LIN {X 0,Y 115.253,Z 407.117,A -85,B 0,C 180,E1 -25932.672,E2 -25932.672} C_VEL
LIN {X 0,Y 115.008,Z 407.148,A -85,B 0,C 180,E1 -25937.79,E2 -25937.79} C_VEL
LIN {X 0,Y 114.944,Z 407.16,A -85,B 0,C 180,E1 -25943.492,E2 -25943.492} C_VEL
LIN {X 0,Y 114.866,Z 407.178,A -85,B 0,C 180,E1 -25946.088,E2 -25946.088} C_VEL
LIN {X 0,Y 115.76,Z 409.771,A -85,B 0,C 180,E1 -25947.086,E2 -25947.086} C_VEL
LIN {X 0,Y 117.751,Z 412.046,A -85,B 0,C 180,E1 -25948.695,E2 -25948.695} C_VEL
LIN {X 0,Y 118.702,Z 412.889,A -85,B 0,C 180,E1 -25949.4,E2 -25949.4} C_VEL
LIN {X 0,Y 120.73,Z 416.135,A -85,B 0,C 180,E1 -25950.969,E2 -25950.969} C_VEL
LIN {X 0,Y 122.361,Z 417.964,A -85,B 0,C 180,E1 -25952.092,E2 -25952.092} C_VEL
LIN {X 0,Y 128.066,Z 426.389,A -85,B 0,C 180,E1 -25955.788,E2 -25955.788} C_VEL
LIN {X 0,Y 130.824,Z 431.068,A -85,B 0,C 180,E1 -25957.424,E2 -25957.424} C_VEL
LIN {X 0,Y 135.904,Z 442.797,A -85,B 0,C 180,E1 -25960.392,E2 -25960.392} C_VEL
LIN {X 0,Y 139.945,Z 454.557,A -85,B 0,C 180,E1 -25962.684,E2 -25962.684} C_VEL
LIN {X 0,Y 140.862,Z 457.48,A -85,B 0,C 180,E1 -25963.193,E2 -25963.193} C_VEL
LIN {X 0,Y 141.678,Z 474.746,A -85,B 0,C 180,E1 -25964.592,E2 -25964.592} C_VEL
LIN {X 0,Y 139.119,Z 511.457,A -85,B 0,C 180,E1 -25966.251,E2 -25966.251} C_VEL
LIN {X 0,Y 137.344,Z 525.013,A -85,B 0,C 180,E1 -25967.355,E2 -25967.355} C_VEL
LIN {X 0,Y 134.916,Z 537.503,A -85,B 0,C 180,E1 -25968.88,E2 -25968.88} C_VEL
LIN {X 0,Y 132.501,Z 547.084,A -85,B 0,C 180,E1 -25970.47,E2 -25970.47} C_VEL
LIN {X 0,Y 129.221,Z 557.848,A -85,B 0,C 180,E1 -25972.768,E2 -25972.768} C_VEL
LIN {X 0,Y 126.712,Z 565.45,A -85,B 0,C 180,E1 -25974.87,E2 -25974.87} C_VEL
LIN {X 0,Y 123.341,Z 575.06,A -85,B 0,C 180,E1 -25978.193,E2 -25978.193} C_VEL
LIN {X 0,Y 119.874,Z 583.772,A -85,B 0,C 180,E1 -25982.03,E2 -25982.03} C_VEL
LIN {X 0,Y 117.346,Z 591.006,A -85,B 0,C 180,E1 -25986.156,E2 -25986.156} C_VEL
LIN {X 0,Y 114.881,Z 598.038,A -85,B 0,C 180,E1 -25991.266,E2 -25991.266} C_VEL
LIN {X 0,Y 113.15,Z 604.474,A -85,B 0,C 180,E1 -25997.444,E2 -25997.444} C_VEL
LIN {X 0,Y 112.538,Z 608.664,A -85,B 0,C 180,E1 -26002.825,E2 -26002.825} C_VEL
LIN {X 0,Y 112.496,Z 611.794,A -85,B 0,C 180,E1 -26008.312,E2 -26008.312} C_VEL
LIN {X 0,Y 112.529,Z 613.372,A -85,B 0,C 180,E1 -26012.193,E2 -26012.193} C_VEL
LIN {X 0,Y 112.474,Z 614.612,A -85,B 0,C 180,E1 -26017.179,E2 -26017.179} C_VEL
LIN {X 0,Y 112.828,Z 615.053,A -85,B 0,C 180,E1 -26020.77,E2 -26020.77} C_VEL
LIN {X 0,Y 114.707,Z 614.724,A -85,B 0,C 180,E1 -26027.839,E2 -26027.839} C_VEL
LIN {X 0,Y 118.407,Z 612.906,A -85,B 0,C 180,E1 -26034.549,E2 -26034.549} C_VEL
LIN {X 0,Y 120.829,Z 611.384,A -85,B 0,C 180,E1 -26037.73,E2 -26037.73} C_VEL
LIN {X 0,Y 125.198,Z 608.337,A -85,B 0,C 180,E1 -26042.227,E2 -26042.227} C_VEL
LIN {X 0,Y 130.219,Z 604.271,A -85,B 0,C 180,E1 -26046.417,E2 -26046.417} C_VEL
LIN {X 0,Y 136.995,Z 598.08,A -85,B 0,C 180,E1 -26050.849,E2 -26050.849} C_VEL
LIN {X 0,Y 143.504,Z 591.376,A -85,B 0,C 180,E1 -26054.256,E2 -26054.256} C_VEL
LIN {X 0,Y 150.582,Z 583.094,A -85,B 0,C 180,E1 -26057.313,E2 -26057.313} C_VEL
LIN {X 0,Y 157.336,Z 573.799,A -85,B 0,C 180,E1 -26059.829,E2 -26059.829} C_VEL
LIN {X 0,Y 159.711,Z 569.48,A -85,B 0,C 180,E1 -26060.999,E2 -26060.999} C_VEL
LIN {X 0,Y 162.549,Z 562.182,A -85,B 0,C 180,E1 -26063.181,E2 -26063.181} C_VEL
LIN {X 0,Y 165.228,Z 554.511,A -85,B 0,C 180,E1 -26065.144,E2 -26065.144} C_VEL
LIN {X 0,Y 167.258,Z 549.517,A -85,B 0,C 180,E1 -26065.962,E2 -26065.962} C_VEL
LIN {X 0,Y 171.699,Z 538.632,A -85,B 0,C 180,E1 -26067.044,E2 -26067.044} C_VEL
LIN {X 0,Y 175.674,Z 525.948,A -85,B 0,C 180,E1 -26067.969,E2 -26067.969} C_VEL
LIN {X 0,Y 178.474,Z 513.103,A -85,B 0,C 180,E1 -26068.575,E2 -26068.575} C_VEL
LIN {X 0,Y 180.148,Z 498.961,A -85,B 0,C 180,E1 -26069.084,E2 -26069.084} C_VEL
LIN {X 0,Y 177.319,Z 490.638,A -85,B 0,C 180,E1 -26072.157,E2 -26072.157} C_VEL
LIN {X 0,Y 175.145,Z 484.92,A -85,B 0,C 180,E1 -26074.844,E2 -26074.844} C_VEL
LIN {X 0,Y 173.289,Z 480.416,A -85,B 0,C 180,E1 -26077.496,E2 -26077.496} C_VEL
LIN {X 0,Y 172.175,Z 477.636,A -85,B 0,C 180,E1 -26079.409,E2 -26079.409} C_VEL
LIN {X 0,Y 170.647,Z 473.807,A -85,B 0,C 180,E1 -26082.724,E2 -26082.724} C_VEL
LIN {X 0,Y 168.918,Z 469.43,A -85,B 0,C 180,E1 -26089.548,E2 -26089.548} C_VEL
LIN {X 0,Y 169.073,Z 469.433,A -85,B 0,C 180,E1 -26096.032,E2 -26096.032} C_VEL
LIN {X 0,Y 170.368,Z 472.982,A -85,B 0,C 180,E1 -26101.182,E2 -26101.182} C_VEL
LIN {X 0,Y 171.205,Z 474.143,A -85,B 0,C 180,E1 -26103.053,E2 -26103.053} C_VEL
LIN {X 0,Y 173.451,Z 478.47,A -85,B 0,C 180,E1 -26107.09,E2 -26107.09} C_VEL
LIN {X 0,Y 175.519,Z 482.29,A -85,B 0,C 180,E1 -26109.871,E2 -26109.871} C_VEL
LIN {X 0,Y 177.675,Z 486.397,A -85,B 0,C 180,E1 -26112.348,E2 -26112.348} C_VEL
LIN {X 0,Y 180.685,Z 492.68,A -85,B 0,C 180,E1 -26115.367,E2 -26115.367} C_VEL
LIN {X 0,Y 178.925,Z 507.485,A -85,B 0,C 180,E1 -26115.96,E2 -26115.96} C_VEL
LIN {X 0,Y 176.106,Z 520.316,A -85,B 0,C 180,E1 -26116.712,E2 -26116.712} C_VEL
LIN {X 0,Y 172.039,Z 533.167,A -85,B 0,C 180,E1 -26117.764,E2 -26117.764} C_VEL
LIN {X 0,Y 167.387,Z 544.658,A -85,B 0,C 180,E1 -26119.152,E2 -26119.152} C_VEL
LIN {X 0,Y 161.724,Z 555.648,A -85,B 0,C 180,E1 -26120.885,E2 -26120.885} C_VEL
LIN {X 0,Y 155.509,Z 565.605,A -85,B 0,C 180,E1 -26122.957,E2 -26122.957} C_VEL
LIN {X 0,Y 149.551,Z 573.711,A -85,B 0,C 180,E1 -26125.184,E2 -26125.184} C_VEL
LIN {X 0,Y 143.124,Z 581.245,A -85,B 0,C 180,E1 -26127.889,E2 -26127.889} C_VEL
LIN {X 0,Y 137.04,Z 587.443,A -85,B 0,C 180,E1 -26130.855,E2 -26130.855} C_VEL
LIN {X 0,Y 131.424,Z 592.438,A -85,B 0,C 180,E1 -26134.019,E2 -26134.019} C_VEL
LIN {X 0,Y 125.209,Z 597.266,A -85,B 0,C 180,E1 -26138.205,E2 -26138.205} C_VEL
LIN {X 0,Y 119.698,Z 600.886,A -85,B 0,C 180,E1 -26142.784,E2 -26142.784} C_VEL
LIN {X 0,Y 114.942,Z 603.398,A -85,B 0,C 180,E1 -26147.734,E2 -26147.734} C_VEL
LIN {X 0,Y 112.305,Z 604.491,A -85,B 0,C 180,E1 -26151.261,E2 -26151.261} C_VEL
LIN {X 0,Y 109.04,Z 605.323,A -85,B 0,C 180,E1 -26156.921,E2 -26156.921} C_VEL
LIN {X 0,Y 106.781,Z 605.183,A -85,B 0,C 180,E1 -26162.567,E2 -26162.567} C_VEL
LIN {X 0,Y 105.395,Z 603.928,A -85,B 0,C 180,E1 -26169,E2 -26169} C_VEL
LIN {X 0,Y 104.928,Z 602.013,A -85,B 0,C 180,E1 -26174.46,E2 -26174.46} C_VEL
LIN {X 0,Y 105.341,Z 598.939,A -85,B 0,C 180,E1 -26180.399,E2 -26180.399} C_VEL
LIN {X 0,Y 106.568,Z 594.793,A -85,B 0,C 180,E1 -26186.219,E2 -26186.219} C_VEL
LIN {X 0,Y 108.751,Z 588.456,A -85,B 0,C 180,E1 -26192.778,E2 -26192.778} C_VEL
LIN {X 0,Y 111.475,Z 581.569,A -85,B 0,C 180,E1 -26198.155,E2 -26198.155} C_VEL
LIN {X 0,Y 114.368,Z 574.542,A -85,B 0,C 180,E1 -26202.42,E2 -26202.42} C_VEL
LIN {X 0,Y 117.794,Z 565.906,A -85,B 0,C 180,E1 -26206.552,E2 -26206.552} C_VEL
LIN {X 0,Y 121.146,Z 556.837,A -85,B 0,C 180,E1 -26209.927,E2 -26209.927} C_VEL
LIN {X 0,Y 125.019,Z 545.291,A -85,B 0,C 180,E1 -26213.172,E2 -26213.172} C_VEL
LIN {X 0,Y 128.216,Z 533.972,A -85,B 0,C 180,E1 -26215.572,E2 -26215.572} C_VEL
LIN {X 0,Y 130.805,Z 522.488,A -85,B 0,C 180,E1 -26217.39,E2 -26217.39} C_VEL
LIN {X 0,Y 133.005,Z 509.199,A -85,B 0,C 180,E1 -26218.844,E2 -26218.844} C_VEL
LIN {X 0,Y 134.384,Z 495.992,A -85,B 0,C 180,E1 -26219.741,E2 -26219.741} C_VEL
LIN {X 0,Y 137.172,Z 456.576,A -85,B 0,C 180,E1 -26221.49,E2 -26221.49} C_VEL
LIN {X 0,Y 131.241,Z 443.73,A -85,B 0,C 180,E1 -26224.758,E2 -26224.758} C_VEL
LIN {X 0,Y 125.369,Z 433.254,A -85,B 0,C 180,E1 -26228.294,E2 -26228.294} C_VEL
LIN {X 0,Y 120.436,Z 425.822,A -85,B 0,C 180,E1 -26231.61,E2 -26231.61} C_VEL
LIN {X 0,Y 118.211,Z 422.576,A -85,B 0,C 180,E1 -26233.267,E2 -26233.267} C_VEL
LIN {X 0,Y 115.739,Z 419.077,A -85,B 0,C 180,E1 -26235.249,E2 -26235.249} C_VEL
LIN {X 0,Y 112.788,Z 415.592,A -85,B 0,C 180,E1 -26237.794,E2 -26237.794} C_VEL
LIN {X 0,Y 111.683,Z 413.593,A -85,B 0,C 180,E1 -26238.914,E2 -26238.914} C_VEL
LIN {X 0,Y 109.275,Z 411.704,A -85,B 0,C 180,E1 -26241.243,E2 -26241.243} C_VEL
LIN {X 0,Y 108.072,Z 409.461,A -85,B 0,C 180,E1 -26242.688,E2 -26242.688} C_VEL
LIN {X 0,Y 107.728,Z 408.052,A -85,B 0,C 180,E1 -26243.368,E2 -26243.368} C_VEL
LIN {X 0,Y 107.799,Z 408.044,A -85,B 0,C 180,E1 -26248.562,E2 -26248.562} C_VEL
LIN {X 0,Y 107.91,Z 408.028,A -85,B 0,C 180,E1 -26256.996,E2 -26256.996} C_VEL
LIN {X 0,Y 108.027,Z 408.014,A -85,B 0,C 180,E1 -26264.915,E2 -26264.915} C_VEL
LIN {X 0,Y 108.254,Z 407.99,A -85,B 0,C 180,E1 -26268.768,E2 -26268.768} C_VEL
LIN {X 0,Y 108.444,Z 407.964,A -85,B 0,C 180,E1 -26276.283,E2 -26276.283} C_VEL
LIN {X 0,Y 108.915,Z 407.86,A -85,B 0,C 180,E1 -26279.999,E2 -26279.999} C_VEL
LIN {X 0,Y 108.301,Z 407.991,A -85,B 0,C 180,E1 -26287.456,E2 -26287.456} C_VEL
LIN {X 0,Y 108.173,Z 408,A -85,B 0,C 180,E1 -26292.959,E2 -26292.959} C_VEL
LIN {X 0,Y 107.943,Z 408.218,A -85,B 0,C 180,E1 -26300.359,E2 -26300.359} C_VEL
LIN {X 0,Y 108.73,Z 410.548,A -85,B 0,C 180,E1 -26301.444,E2 -26301.444} C_VEL
LIN {X 0,Y 110.675,Z 412.834,A -85,B 0,C 180,E1 -26303.485,E2 -26303.485} C_VEL
LIN {X 0,Y 112.053,Z 413.96,A -85,B 0,C 180,E1 -26304.763,E2 -26304.763} C_VEL
LIN {X 0,Y 114.154,Z 417.301,A -85,B 0,C 180,E1 -26306.756,E2 -26306.756} C_VEL
LIN {X 0,Y 115.855,Z 419.178,A -85,B 0,C 180,E1 -26308.165,E2 -26308.165} C_VEL
LIN {X 0,Y 118.456,Z 422.775,A -85,B 0,C 180,E1 -26310.232,E2 -26310.232} C_VEL
LIN {X 0,Y 122.616,Z 428.986,A -85,B 0,C 180,E1 -26313.236,E2 -26313.236} C_VEL
LIN {X 0,Y 126.523,Z 435.357,A -85,B 0,C 180,E1 -26315.786,E2 -26315.786} C_VEL
LIN {X 0,Y 131.342,Z 446.96,A -85,B 0,C 180,E1 -26318.864,E2 -26318.864} C_VEL
LIN {X 0,Y 135.02,Z 458.215,A -85,B 0,C 180,E1 -26321.159,E2 -26321.159} C_VEL
LIN {X 0,Y 135.529,Z 460.494,A -85,B 0,C 180,E1 -26321.512,E2 -26321.512} C_VEL
LIN {X 0,Y 136.182,Z 474.785,A -85,B 0,C 180,E1 -26322.748,E2 -26322.748} C_VEL
LIN {X 0,Y 133.574,Z 510.886,A -85,B 0,C 180,E1 -26324.416,E2 -26324.416} C_VEL
LIN {X 0,Y 131.674,Z 524.54,A -85,B 0,C 180,E1 -26325.531,E2 -26325.531} C_VEL
LIN {X 0,Y 129.103,Z 537.266,A -85,B 0,C 180,E1 -26327.121,E2 -26327.121} C_VEL
LIN {X 0,Y 126.576,Z 546.828,A -85,B 0,C 180,E1 -26328.751,E2 -26328.751} C_VEL
LIN {X 0,Y 123.147,Z 557.577,A -85,B 0,C 180,E1 -26331.115,E2 -26331.115} C_VEL
LIN {X 0,Y 120.493,Z 565.166,A -85,B 0,C 180,E1 -26333.285,E2 -26333.285} C_VEL
LIN {X 0,Y 117.302,Z 573.776,A -85,B 0,C 180,E1 -26336.345,E2 -26336.345} C_VEL
LIN {X 0,Y 114.329,Z 580.973,A -85,B 0,C 180,E1 -26339.503,E2 -26339.503} C_VEL
LIN {X 0,Y 111.365,Z 588.648,A -85,B 0,C 180,E1 -26343.785,E2 -26343.785} C_VEL
LIN {X 0,Y 108.54,Z 596.111,A -85,B 0,C 180,E1 -26349.138,E2 -26349.138} C_VEL
LIN {X 0,Y 106.591,Z 602.073,A -85,B 0,C 180,E1 -26354.708,E2 -26354.708} C_VEL
LIN {X 0,Y 105.642,Z 606.757,A -85,B 0,C 180,E1 -26360.426,E2 -26360.426} C_VEL
LIN {X 0,Y 105.39,Z 610.28,A -85,B 0,C 180,E1 -26366.176,E2 -26366.176} C_VEL
LIN {X 0,Y 105.548,Z 612.037,A -85,B 0,C 180,E1 -26370,E2 -26370} C_VEL
LIN {X 0,Y 105.389,Z 613.311,A -85,B 0,C 180,E1 -26373.824,E2 -26373.824} C_VEL
LIN {X 0,Y 105.834,Z 614.67,A -85,B 0,C 180,E1 -26381.491,E2 -26381.491} C_VEL
LIN {X 0,Y 106.688,Z 614.76,A -85,B 0,C 180,E1 -26385.277,E2 -26385.277} C_VEL
LIN {X 0,Y 109.705,Z 613.761,A -85,B 0,C 180,E1 -26392.605,E2 -26392.605} C_VEL
LIN {X 0,Y 114.575,Z 611.256,A -85,B 0,C 180,E1 -26399.387,E2 -26399.387} C_VEL
LIN {X 0,Y 119.817,Z 607.841,A -85,B 0,C 180,E1 -26404.603,E2 -26404.603} C_VEL
LIN {X 0,Y 126.503,Z 602.701,A -85,B 0,C 180,E1 -26409.708,E2 -26409.708} C_VEL
LIN {X 0,Y 133.931,Z 596.208,A -85,B 0,C 180,E1 -26414.049,E2 -26414.049} C_VEL
LIN {X 0,Y 140.938,Z 589.139,A -85,B 0,C 180,E1 -26417.35,E2 -26417.35} C_VEL
LIN {X 0,Y 148.421,Z 580.361,A -85,B 0,C 180,E1 -26420.305,E2 -26420.305} C_VEL
LIN {X 0,Y 155.615,Z 570.432,A -85,B 0,C 180,E1 -26422.747,E2 -26422.747} C_VEL
LIN {X 0,Y 161.818,Z 560.324,A -85,B 0,C 180,E1 -26424.52,E2 -26424.52} C_VEL
LIN {X 0,Y 167.258,Z 549.517,A -85,B 0,C 180,E1 -26425.962,E2 -26425.962} C_VEL
LIN {X 0,Y 169.166,Z 544.407,A -85,B 0,C 180,E1 -26426.717,E2 -26426.717} C_VEL
LIN {X 0,Y 171.161,Z 535.908,A -85,B 0,C 180,E1 -26428.307,E2 -26428.307} C_VEL
LIN {X 0,Y 172.711,Z 527.169,A -85,B 0,C 180,E1 -26429.764,E2 -26429.764} C_VEL
LIN {X 0,Y 173.83,Z 521.619,A -85,B 0,C 180,E1 -26430.314,E2 -26430.314} C_VEL
LIN {X 0,Y 176.309,Z 508.882,A -85,B 0,C 180,E1 -26430.844,E2 -26430.844} C_VEL
LIN {X 0,Y 177.063,Z 502.166,A -85,B 0,C 180,E1 -26431.088,E2 -26431.088} C_VEL
LIN {X 0,Y 174.716,Z 494.887,A -85,B 0,C 180,E1 -26433.979,E2 -26433.979} C_VEL
LIN {X 0,Y 172.504,Z 488.69,A -85,B 0,C 180,E1 -26437.151,E2 -26437.151} C_VEL
LIN {X 0,Y 170.816,Z 484.212,A -85,B 0,C 180,E1 -26440.165,E2 -26440.165} C_VEL
LIN {X 0,Y 169.455,Z 480.555,A -85,B 0,C 180,E1 -26443.393,E2 -26443.393} C_VEL
LIN {X 0,Y 167.982,Z 476.435,A -85,B 0,C 180,E1 -26449.928,E2 -26449.928} C_VEL
LIN {X 0,Y 168.17,Z 476.581,A -85,B 0,C 180,E1 -26456.011,E2 -26456.011} C_VEL
LIN {X 0,Y 169.126,Z 479.622,A -85,B 0,C 180,E1 -26460.298,E2 -26460.298} C_VEL
LIN {X 0,Y 169.969,Z 480.84,A -85,B 0,C 180,E1 -26462.37,E2 -26462.37} C_VEL
LIN {X 0,Y 172,Z 485.034,A -85,B 0,C 180,E1 -26466.333,E2 -26466.333} C_VEL
LIN {X 0,Y 174.107,Z 489.188,A -85,B 0,C 180,E1 -26469.366,E2 -26469.366} C_VEL
LIN {X 0,Y 177.049,Z 495.311,A -85,B 0,C 180,E1 -26472.83,E2 -26472.83} C_VEL
LIN {X 0,Y 177.618,Z 496.635,A -85,B 0,C 180,E1 -26473.443,E2 -26473.443} C_VEL
LIN {X 0,Y 175.731,Z 509.626,A -85,B 0,C 180,E1 -26473.951,E2 -26473.951} C_VEL
LIN {X 0,Y 172.695,Z 522.371,A -85,B 0,C 180,E1 -26474.708,E2 -26474.708} C_VEL
LIN {X 0,Y 168.729,Z 534.274,A -85,B 0,C 180,E1 -26475.693,E2 -26475.693} C_VEL
LIN {X 0,Y 163.622,Z 546.148,A -85,B 0,C 180,E1 -26477.124,E2 -26477.124} C_VEL
LIN {X 0,Y 157.583,Z 557.253,A -85,B 0,C 180,E1 -26478.872,E2 -26478.872} C_VEL
LIN {X 0,Y 152.044,Z 565.713,A -85,B 0,C 180,E1 -26480.61,E2 -26480.61} C_VEL
LIN {X 0,Y 145.129,Z 574.749,A -85,B 0,C 180,E1 -26483.064,E2 -26483.064} C_VEL
LIN {X 0,Y 138.482,Z 582.111,A -85,B 0,C 180,E1 -26485.737,E2 -26485.737} C_VEL
LIN {X 0,Y 131.112,Z 589.093,A -85,B 0,C 180,E1 -26489.224,E2 -26489.224} C_VEL
LIN {X 0,Y 125.088,Z 594.012,A -85,B 0,C 180,E1 -26492.569,E2 -26492.569} C_VEL
LIN {X 0,Y 118.379,Z 598.69,A -85,B 0,C 180,E1 -26497.085,E2 -26497.085} C_VEL
LIN {X 0,Y 112.898,Z 601.877,A -85,B 0,C 180,E1 -26501.669,E2 -26501.669} C_VEL
LIN {X 0,Y 109.512,Z 603.507,A -85,B 0,C 180,E1 -26505.096,E2 -26505.096} C_VEL
LIN {X 0,Y 106.542,Z 604.699,A -85,B 0,C 180,E1 -26508.728,E2 -26508.728} C_VEL
LIN {X 0,Y 102.488,Z 605.665,A -85,B 0,C 180,E1 -26515.377,E2 -26515.377} C_VEL
LIN {X 0,Y 100.219,Z 605.582,A -85,B 0,C 180,E1 -26520.602,E2 -26520.602} C_VEL
LIN {X 0,Y 98.388,Z 604.245,A -85,B 0,C 180,E1 -26528.223,E2 -26528.223} C_VEL
LIN {X 0,Y 97.865,Z 602.604,A -85,B 0,C 180,E1 -26533.307,E2 -26533.307} C_VEL
LIN {X 0,Y 98.162,Z 599.637,A -85,B 0,C 180,E1 -26539.689,E2 -26539.689} C_VEL
LIN {X 0,Y 99.323,Z 595.612,A -85,B 0,C 180,E1 -26545.943,E2 -26545.943} C_VEL
LIN {X 0,Y 101.176,Z 590.451,A -85,B 0,C 180,E1 -26551.99,E2 -26551.99} C_VEL
LIN {X 0,Y 103.832,Z 583.961,A -85,B 0,C 180,E1 -26557.78,E2 -26557.78} C_VEL
LIN {X 0,Y 107.381,Z 575.844,A -85,B 0,C 180,E1 -26563.242,E2 -26563.242} C_VEL
LIN {X 0,Y 111.167,Z 566.932,A -85,B 0,C 180,E1 -26567.816,E2 -26567.816} C_VEL
LIN {X 0,Y 114.882,Z 557.497,A -85,B 0,C 180,E1 -26571.534,E2 -26571.534} C_VEL
LIN {X 0,Y 118.972,Z 546.031,A -85,B 0,C 180,E1 -26574.89,E2 -26574.89} C_VEL
LIN {X 0,Y 122.312,Z 534.816,A -85,B 0,C 180,E1 -26577.366,E2 -26577.366} C_VEL
LIN {X 0,Y 125.293,Z 522.284,A -85,B 0,C 180,E1 -26579.393,E2 -26579.393} C_VEL
LIN {X 0,Y 127.558,Z 509.173,A -85,B 0,C 180,E1 -26580.834,E2 -26580.834} C_VEL
LIN {X 0,Y 128.99,Z 495.882,A -85,B 0,C 180,E1 -26581.743,E2 -26581.743} C_VEL
LIN {X 0,Y 131.739,Z 458.836,A -85,B 0,C 180,E1 -26583.411,E2 -26583.411} C_VEL
LIN {X 0,Y 126.381,Z 447.016,A -85,B 0,C 180,E1 -26586.66,E2 -26586.66} C_VEL
LIN {X 0,Y 120.783,Z 436.959,A -85,B 0,C 180,E1 -26590.377,E2 -26590.377} C_VEL
LIN {X 0,Y 115.331,Z 428.518,A -85,B 0,C 180,E1 -26594.525,E2 -26594.525} C_VEL
LIN {X 0,Y 112.025,Z 424.051,A -85,B 0,C 180,E1 -26597.399,E2 -26597.399} C_VEL
LIN {X 0,Y 109.54,Z 420.544,A -85,B 0,C 180,E1 -26599.857,E2 -26599.857} C_VEL
LIN {X 0,Y 108.684,Z 419.589,A -85,B 0,C 180,E1 -26600.739,E2 -26600.739} C_VEL
LIN {X 0,Y 106.413,Z 417.142,A -85,B 0,C 180,E1 -26603.254,E2 -26603.254} C_VEL
LIN {X 0,Y 105.258,Z 414.722,A -85,B 0,C 180,E1 -26604.837,E2 -26604.837} C_VEL
LIN {X 0,Y 102.666,Z 412.959,A -85,B 0,C 180,E1 -26608.238,E2 -26608.238} C_VEL
LIN {X 0,Y 101.105,Z 410.644,A -85,B 0,C 180,E1 -26610.883,E2 -26610.883} C_VEL
LIN {X 0,Y 100.692,Z 408.94,A -85,B 0,C 180,E1 -26612.034,E2 -26612.034} C_VEL
LIN {X 0,Y 100.786,Z 408.917,A -85,B 0,C 180,E1 -26615.266,E2 -26615.266} C_VEL
LIN {X 0,Y 100.814,Z 408.926,A -85,B 0,C 180,E1 -26619.599,E2 -26619.599} C_VEL
LIN {X 0,Y 101.102,Z 408.888,A -85,B 0,C 180,E1 -26626.697,E2 -26626.697} C_VEL
LIN {X 0,Y 101.242,Z 408.858,A -85,B 0,C 180,E1 -26632.018,E2 -26632.018} C_VEL
LIN {X 0,Y 101.842,Z 408.739,A -85,B 0,C 180,E1 -26639.999,E2 -26639.999} C_VEL
LIN {X 0,Y 101.24,Z 408.873,A -85,B 0,C 180,E1 -26647.98,E2 -26647.98} C_VEL
LIN {X 0,Y 101.165,Z 408.908,A -85,B 0,C 180,E1 -26652.183,E2 -26652.183} C_VEL
LIN {X 0,Y 101.902,Z 411.444,A -85,B 0,C 180,E1 -26653.772,E2 -26653.772} C_VEL
LIN {X 0,Y 103.665,Z 413.707,A -85,B 0,C 180,E1 -26656.492,E2 -26656.492} C_VEL
LIN {X 0,Y 105.525,Z 414.848,A -85,B 0,C 180,E1 -26658.819,E2 -26658.819} C_VEL
LIN {X 0,Y 107.306,Z 418.07,A -85,B 0,C 180,E1 -26661.113,E2 -26661.113} C_VEL
LIN {X 0,Y 109.51,Z 420.308,A -85,B 0,C 180,E1 -26663.425,E2 -26663.425} C_VEL
LIN {X 0,Y 111.933,Z 423.843,A -85,B 0,C 180,E1 -26665.832,E2 -26665.832} C_VEL
LIN {X 0,Y 113.231,Z 425.595,A -85,B 0,C 180,E1 -26667.007,E2 -26667.007} C_VEL
LIN {X 0,Y 116.505,Z 430.3,A -85,B 0,C 180,E1 -26669.754,E2 -26669.754} C_VEL
LIN {X 0,Y 120.937,Z 437.212,A -85,B 0,C 180,E1 -26673.058,E2 -26673.058} C_VEL
LIN {X 0,Y 122.685,Z 440.49,A -85,B 0,C 180,E1 -26674.294,E2 -26674.294} C_VEL
LIN {X 0,Y 126.846,Z 451.098,A -85,B 0,C 180,E1 -26677.222,E2 -26677.222} C_VEL
LIN {X 0,Y 130.283,Z 462.04,A -85,B 0,C 180,E1 -26679.568,E2 -26679.568} C_VEL
LIN {X 0,Y 130.779,Z 475.55,A -85,B 0,C 180,E1 -26680.782,E2 -26680.782} C_VEL
LIN {X 0,Y 128.064,Z 511.015,A -85,B 0,C 180,E1 -26682.461,E2 -26682.461} C_VEL
LIN {X 0,Y 126.124,Z 524.347,A -85,B 0,C 180,E1 -26683.583,E2 -26683.583} C_VEL
LIN {X 0,Y 123.423,Z 537.028,A -85,B 0,C 180,E1 -26685.199,E2 -26685.199} C_VEL
LIN {X 0,Y 120.765,Z 546.567,A -85,B 0,C 180,E1 -26686.86,E2 -26686.86} C_VEL
LIN {X 0,Y 117.184,Z 557.305,A -85,B 0,C 180,E1 -26689.292,E2 -26689.292} C_VEL
LIN {X 0,Y 114.379,Z 564.883,A -85,B 0,C 180,E1 -26691.529,E2 -26691.529} C_VEL
LIN {X 0,Y 110.612,Z 574.478,A -85,B 0,C 180,E1 -26695.123,E2 -26695.123} C_VEL
LIN {X 0,Y 106.716,Z 583.169,A -85,B 0,C 180,E1 -26699.311,E2 -26699.311} C_VEL
LIN {X 0,Y 103.846,Z 590.396,A -85,B 0,C 180,E1 -26703.903,E2 -26703.903} C_VEL
LIN {X 0,Y 101.033,Z 597.415,A -85,B 0,C 180,E1 -26709.647,E2 -26709.647} C_VEL
LIN {X 0,Y 99.247,Z 603.023,A -85,B 0,C 180,E1 -26715.65,E2 -26715.65} C_VEL
LIN {X 0,Y 98.437,Z 607.399,A -85,B 0,C 180,E1 -26721.791,E2 -26721.791} C_VEL
LIN {X 0,Y 98.309,Z 609.691,A -85,B 0,C 180,E1 -26725.901,E2 -26725.901} C_VEL
LIN {X 0,Y 98.428,Z 612.071,A -85,B 0,C 180,E1 -26731.583,E2 -26731.583} C_VEL
LIN {X 0,Y 98.373,Z 613.749,A -85,B 0,C 180,E1 -26738.215,E2 -26738.215} C_VEL
LIN {X 0,Y 99.812,Z 614.427,A -85,B 0,C 180,E1 -26746.358,E2 -26746.358} C_VEL
LIN {X 0,Y 101.207,Z 614.166,A -85,B 0,C 180,E1 -26750.316,E2 -26750.316} C_VEL
LIN {X 0,Y 105.618,Z 612.503,A -85,B 0,C 180,E1 -26757.761,E2 -26757.761} C_VEL
LIN {X 0,Y 108.431,Z 611.102,A -85,B 0,C 180,E1 -26761.232,E2 -26761.232} C_VEL
LIN {X 0,Y 114.607,Z 607.4,A -85,B 0,C 180,E1 -26767.138,E2 -26767.138} C_VEL
LIN {X 0,Y 121.129,Z 602.775,A -85,B 0,C 180,E1 -26771.853,E2 -26771.853} C_VEL
LIN {X 0,Y 128.933,Z 596.389,A -85,B 0,C 180,E1 -26776.238,E2 -26776.238} C_VEL
LIN {X 0,Y 136.232,Z 589.474,A -85,B 0,C 180,E1 -26779.544,E2 -26779.544} C_VEL
LIN {X 0,Y 144.011,Z 580.857,A -85,B 0,C 180,E1 -26782.468,E2 -26782.468} C_VEL
LIN {X 0,Y 150.749,Z 572.067,A -85,B 0,C 180,E1 -26784.671,E2 -26784.671} C_VEL
LIN {X 0,Y 157.816,Z 561.264,A -85,B 0,C 180,E1 -26786.613,E2 -26786.613} C_VEL
LIN {X 0,Y 163.801,Z 549.976,A -85,B 0,C 180,E1 -26788.095,E2 -26788.095} C_VEL
LIN {X 0,Y 168.717,Z 538.344,A -85,B 0,C 180,E1 -26789.219,E2 -26789.219} C_VEL
LIN {X 0,Y 172.544,Z 526.559,A -85,B 0,C 180,E1 -26790.052,E2 -26790.052} C_VEL
LIN {X 0,Y 173.83,Z 521.619,A -85,B 0,C 180,E1 -26790.314,E2 -26790.314} C_VEL
LIN {X 0,Y 174.637,Z 516.494,A -85,B 0,C 180,E1 -26790.82,E2 -26790.82} C_VEL
LIN {X 0,Y 174.748,Z 511.664,A -85,B 0,C 180,E1 -26791.634,E2 -26791.634} C_VEL
LIN {X 0,Y 174.361,Z 507.256,A -85,B 0,C 180,E1 -26792.7,E2 -26792.7} C_VEL
LIN {X 0,Y 173.577,Z 503.433,A -85,B 0,C 180,E1 -26793.971,E2 -26793.971} C_VEL
LIN {X 0,Y 171.583,Z 497.126,A -85,B 0,C 180,E1 -26796.941,E2 -26796.941} C_VEL
LIN {X 0,Y 170.098,Z 492.743,A -85,B 0,C 180,E1 -26799.598,E2 -26799.598} C_VEL
LIN {X 0,Y 169.338,Z 490.475,A -85,B 0,C 180,E1 -26801.247,E2 -26801.247} C_VEL
LIN {X 0,Y 168.284,Z 487.277,A -85,B 0,C 180,E1 -26804.086,E2 -26804.086} C_VEL
LIN {X 0,Y 167.054,Z 483.44,A -85,B 0,C 180,E1 -26810.313,E2 -26810.313} C_VEL
LIN {X 0,Y 167.197,Z 483.527,A -85,B 0,C 180,E1 -26815.48,E2 -26815.48} C_VEL
LIN {X 0,Y 168.329,Z 486.931,A -85,B 0,C 180,E1 -26820.599,E2 -26820.599} C_VEL
LIN {X 0,Y 168.914,Z 487.971,A -85,B 0,C 180,E1 -26822.094,E2 -26822.094} C_VEL
LIN {X 0,Y 170.641,Z 491.747,A -85,B 0,C 180,E1 -26825.67,E2 -26825.67} C_VEL
LIN {X 0,Y 172.707,Z 496.101,A -85,B 0,C 180,E1 -26828.852,E2 -26828.852} C_VEL
LIN {X 0,Y 174.628,Z 500.536,A -85,B 0,C 180,E1 -26831.398,E2 -26831.398} C_VEL
LIN {X 0,Y 172.416,Z 513.478,A -85,B 0,C 180,E1 -26831.968,E2 -26831.968} C_VEL
LIN {X 0,Y 169.134,Z 525.575,A -85,B 0,C 180,E1 -26832.719,E2 -26832.719} C_VEL
LIN {X 0,Y 164.632,Z 537.775,A -85,B 0,C 180,E1 -26833.795,E2 -26833.795} C_VEL
LIN {X 0,Y 159.247,Z 549.261,A -85,B 0,C 180,E1 -26835.225,E2 -26835.225} C_VEL
LIN {X 0,Y 153.299,Z 559.4,A -85,B 0,C 180,E1 -26836.865,E2 -26836.865} C_VEL
LIN {X 0,Y 146.681,Z 568.75,A -85,B 0,C 180,E1 -26838.87,E2 -26838.87} C_VEL
LIN {X 0,Y 139.554,Z 577.244,A -85,B 0,C 180,E1 -26841.308,E2 -26841.308} C_VEL
LIN {X 0,Y 131.381,Z 585.492,A -85,B 0,C 180,E1 -26844.582,E2 -26844.582} C_VEL
LIN {X 0,Y 123.67,Z 591.971,A -85,B 0,C 180,E1 -26848.258,E2 -26848.258} C_VEL
LIN {X 0,Y 116.534,Z 597.047,A -85,B 0,C 180,E1 -26852.403,E2 -26852.403} C_VEL
LIN {X 0,Y 110.043,Z 600.893,A -85,B 0,C 180,E1 -26857.032,E2 -26857.032} C_VEL
LIN {X 0,Y 104.018,Z 603.753,A -85,B 0,C 180,E1 -26862.506,E2 -26862.506} C_VEL
LIN {X 0,Y 101.028,Z 604.874,A -85,B 0,C 180,E1 -26865.923,E2 -26865.923} C_VEL
LIN {X 0,Y 98.178,Z 605.68,A -85,B 0,C 180,E1 -26869.891,E2 -26869.891} C_VEL
LIN {X 0,Y 95.784,Z 606.021,A -85,B 0,C 180,E1 -26874.057,E2 -26874.057} C_VEL
LIN {X 0,Y 93.807,Z 605.957,A -85,B 0,C 180,E1 -26878.37,E2 -26878.37} C_VEL
LIN {X 0,Y 92.339,Z 605.484,A -85,B 0,C 180,E1 -26882.829,E2 -26882.829} C_VEL
LIN {X 0,Y 91.403,Z 604.542,A -85,B 0,C 180,E1 -26887.391,E2 -26887.391} C_VEL
LIN {X 0,Y 90.857,Z 603.187,A -85,B 0,C 180,E1 -26891.977,E2 -26891.977} C_VEL
LIN {X 0,Y 90.974,Z 600.331,A -85,B 0,C 180,E1 -26898.865,E2 -26898.865} C_VEL
LIN {X 0,Y 92.06,Z 596.424,A -85,B 0,C 180,E1 -26905.622,E2 -26905.622} C_VEL
LIN {X 0,Y 93.997,Z 591.378,A -85,B 0,C 180,E1 -26912.142,E2 -26912.142} C_VEL
LIN {X 0,Y 96.719,Z 585.059,A -85,B 0,C 180,E1 -26918.356,E2 -26918.356} C_VEL
LIN {X 0,Y 100.445,Z 577.142,A -85,B 0,C 180,E1 -26924.175,E2 -26924.175} C_VEL
LIN {X 0,Y 104.911,Z 567.266,A -85,B 0,C 180,E1 -26929.569,E2 -26929.569} C_VEL
LIN {X 0,Y 108.72,Z 558.146,A -85,B 0,C 180,E1 -26933.324,E2 -26933.324} C_VEL
LIN {X 0,Y 113.027,Z 546.777,A -85,B 0,C 180,E1 -26936.795,E2 -26936.795} C_VEL
LIN {X 0,Y 116.551,Z 535.656,A -85,B 0,C 180,E1 -26939.335,E2 -26939.335} C_VEL
LIN {X 0,Y 119.674,Z 523.335,A -85,B 0,C 180,E1 -26941.412,E2 -26941.412} C_VEL
LIN {X 0,Y 122.083,Z 510.375,A -85,B 0,C 180,E1 -26942.893,E2 -26942.893} C_VEL
LIN {X 0,Y 123.678,Z 496.64,A -85,B 0,C 180,E1 -26943.871,E2 -26943.871} C_VEL
LIN {X 0,Y 126.435,Z 460.997,A -85,B 0,C 180,E1 -26945.507,E2 -26945.507} C_VEL
LIN {X 0,Y 121.689,Z 450.503,A -85,B 0,C 180,E1 -26948.675,E2 -26948.675} C_VEL
LIN {X 0,Y 116.68,Z 441.262,A -85,B 0,C 180,E1 -26952.358,E2 -26952.358} C_VEL
LIN {X 0,Y 112.101,Z 434.027,A -85,B 0,C 180,E1 -26956.2,E2 -26956.2} C_VEL
LIN {X 0,Y 108.937,Z 429.523,A -85,B 0,C 180,E1 -26959.239,E2 -26959.239} C_VEL
LIN {X 0,Y 106.502,Z 426.035,A -85,B 0,C 180,E1 -26961.91,E2 -26961.91} C_VEL
LIN {X 0,Y 104.02,Z 423.093,A -85,B 0,C 180,E1 -26964.912,E2 -26964.912} C_VEL
LIN {X 0,Y 103.076,Z 421.255,A -85,B 0,C 180,E1 -26966.298,E2 -26966.298} C_VEL
LIN {X 0,Y 100.425,Z 418.94,A -85,B 0,C 180,E1 -26970.233,E2 -26970.233} C_VEL
LIN {X 0,Y 99.003,Z 416.252,A -85,B 0,C 180,E1 -26973.091,E2 -26973.091} C_VEL
LIN {X 0,Y 98.784,Z 415.762,A -85,B 0,C 180,E1 -26973.597,E2 -26973.597} C_VEL
LIN {X 0,Y 95.396,Z 413.449,A -85,B 0,C 180,E1 -26982.86,E2 -26982.86} C_VEL
LIN {X 0,Y 94.673,Z 411.791,A -85,B 0,C 180,E1 -26988.219,E2 -26988.219} C_VEL
LIN {X 0,Y 94.564,Z 411.328,A -85,B 0,C 180,E1 -26991.451,E2 -26991.451} C_VEL
LIN {X 0,Y 95.514,Z 412.079,A -85,B 0,C 180,E1 -27000.262,E2 -27000.262} C_VEL
LIN {X 0,Y 96.64,Z 414.177,A -85,B 0,C 180,E1 -27004.692,E2 -27004.692} C_VEL
LIN {X 0,Y 99.322,Z 415.889,A -85,B 0,C 180,E1 -27010.704,E2 -27010.704} C_VEL
LIN {X 0,Y 100.544,Z 418.685,A -85,B 0,C 180,E1 -27013.223,E2 -27013.223} C_VEL
LIN {X 0,Y 102.582,Z 420.839,A -85,B 0,C 180,E1 -27016.363,E2 -27016.363} C_VEL
LIN {X 0,Y 103.441,Z 421.546,A -85,B 0,C 180,E1 -27017.521,E2 -27017.521} C_VEL
LIN {X 0,Y 105.628,Z 424.993,A -85,B 0,C 180,E1 -27020.428,E2 -27020.428} C_VEL
LIN {X 0,Y 107.089,Z 426.612,A -85,B 0,C 180,E1 -27022.074,E2 -27022.074} C_VEL
LIN {X 0,Y 109.684,Z 430.31,A -85,B 0,C 180,E1 -27024.813,E2 -27024.813} C_VEL
LIN {X 0,Y 114.928,Z 438.276,A -85,B 0,C 180,E1 -27029.549,E2 -27029.549} C_VEL
LIN {X 0,Y 118.535,Z 444.605,A -85,B 0,C 180,E1 -27032.391,E2 -27032.391} C_VEL
LIN {X 0,Y 122.454,Z 455.134,A -85,B 0,C 180,E1 -27035.449,E2 -27035.449} C_VEL
LIN {X 0,Y 125.228,Z 464.515,A -85,B 0,C 180,E1 -27037.565,E2 -27037.565} C_VEL
LIN {X 0,Y 125.581,Z 475.817,A -85,B 0,C 180,E1 -27038.629,E2 -27038.629} C_VEL
LIN {X 0,Y 122.767,Z 510.797,A -85,B 0,C 180,E1 -27040.312,E2 -27040.312} C_VEL
LIN {X 0,Y 120.716,Z 524.138,A -85,B 0,C 180,E1 -27041.448,E2 -27041.448} C_VEL
LIN {X 0,Y 117.895,Z 536.789,A -85,B 0,C 180,E1 -27043.094,E2 -27043.094} C_VEL
LIN {X 0,Y 115.109,Z 546.311,A -85,B 0,C 180,E1 -27044.786,E2 -27044.786} C_VEL
LIN {X 0,Y 111.349,Z 557.032,A -85,B 0,C 180,E1 -27047.274,E2 -27047.274} C_VEL
LIN {X 0,Y 108.386,Z 564.601,A -85,B 0,C 180,E1 -27049.578,E2 -27049.578} C_VEL
LIN {X 0,Y 104.214,Z 574.633,A -85,B 0,C 180,E1 -27053.508,E2 -27053.508} C_VEL
LIN {X 0,Y 99.816,Z 583.927,A -85,B 0,C 180,E1 -27058.352,E2 -27058.352} C_VEL
LIN {X 0,Y 96.905,Z 590.723,A -85,B 0,C 180,E1 -27063.046,E2 -27063.046} C_VEL
LIN {X 0,Y 93.938,Z 597.615,A -85,B 0,C 180,E1 -27069.184,E2 -27069.184} C_VEL
LIN {X 0,Y 91.914,Z 603.935,A -85,B 0,C 180,E1 -27076.739,E2 -27076.739} C_VEL
LIN {X 0,Y 91.249,Z 608.013,A -85,B 0,C 180,E1 -27083.366,E2 -27083.366} C_VEL
LIN {X 0,Y 91.37,Z 611.246,A -85,B 0,C 180,E1 -27090.701,E2 -27090.701} C_VEL
LIN {X 0,Y 91.215,Z 612.372,A -85,B 0,C 180,E1 -27094.419,E2 -27094.419} C_VEL
LIN {X 0,Y 91.938,Z 613.884,A -85,B 0,C 180,E1 -27103.257,E2 -27103.257} C_VEL
LIN {X 0,Y 94.548,Z 613.883,A -85,B 0,C 180,E1 -27111.818,E2 -27111.818} C_VEL
LIN {X 0,Y 99.357,Z 612.31,A -85,B 0,C 180,E1 -27119.678,E2 -27119.678} C_VEL
LIN {X 0,Y 105.874,Z 609.203,A -85,B 0,C 180,E1 -27126.685,E2 -27126.685} C_VEL
LIN {X 0,Y 111.649,Z 605.735,A -85,B 0,C 180,E1 -27131.371,E2 -27131.371} C_VEL
LIN {X 0,Y 118.18,Z 601.229,A -85,B 0,C 180,E1 -27135.529,E2 -27135.529} C_VEL
LIN {X 0,Y 126.591,Z 594.469,A -85,B 0,C 180,E1 -27139.76,E2 -27139.76} C_VEL
LIN {X 0,Y 134.368,Z 587.15,A -85,B 0,C 180,E1 -27142.903,E2 -27142.903} C_VEL
LIN {X 0,Y 142.595,Z 578.104,A -85,B 0,C 180,E1 -27145.642,E2 -27145.642} C_VEL
LIN {X 0,Y 149.65,Z 568.778,A -85,B 0,C 180,E1 -27147.706,E2 -27147.706} C_VEL
LIN {X 0,Y 156.234,Z 558.442,A -85,B 0,C 180,E1 -27149.35,E2 -27149.35} C_VEL
LIN {X 0,Y 162.223,Z 546.993,A -85,B 0,C 180,E1 -27150.675,E2 -27150.675} C_VEL
LIN {X 0,Y 167.11,Z 535.041,A -85,B 0,C 180,E1 -27151.706,E2 -27151.706} C_VEL
LIN {X 0,Y 171.145,Z 521.702,A -85,B 0,C 180,E1 -27152.488,E2 -27152.488} C_VEL
LIN {X 0,Y 173.77,Z 508.635,A -85,B 0,C 180,E1 -27153.018,E2 -27153.018} C_VEL
LIN {X 0,Y 174.09,Z 505.387,A -85,B 0,C 180,E1 -27153.207,E2 -27153.207} C_VEL
LIN {X 0,Y 173.577,Z 503.433,A -85,B 0,C 180,E1 -27153.971,E2 -27153.971} C_VEL
LIN {X 0,Y 172.824,Z 501.326,A -85,B 0,C 180,E1 -27155.035,E2 -27155.035} C_VEL
LIN {X 0,Y 171.46,Z 499.344,A -85,B 0,C 180,E1 -27156.837,E2 -27156.837} C_VEL
LIN {X 0,Y 168.413,Z 497.044,A -85,B 0,C 180,E1 -27161.436,E2 -27161.436} C_VEL
LIN {X 0,Y 167.554,Z 495.451,A -85,B 0,C 180,E1 -27163.413,E2 -27163.413} C_VEL
LIN {X 0,Y 167.366,Z 494.654,A -85,B 0,C 180,E1 -27164.046,E2 -27164.046} C_VEL
LIN {X 0,Y 166.46,Z 492.422,A -85,B 0,C 180,E1 -27167.455,E2 -27167.455} C_VEL
LIN {X 0,Y 166.116,Z 490.46,A -85,B 0,C 180,E1 -27170.872,E2 -27170.872} C_VEL
LIN {X 0,Y 166.277,Z 490.606,A -85,B 0,C 180,E1 -27175.303,E2 -27175.303} C_VEL
LIN {X 0,Y 167.281,Z 493.857,A -85,B 0,C 180,E1 -27180.204,E2 -27180.204} C_VEL
LIN {X 0,Y 167.755,Z 494.799,A -85,B 0,C 180,E1 -27181.518,E2 -27181.518} C_VEL
LIN {X 0,Y 169.277,Z 498.338,A -85,B 0,C 180,E1 -27184.932,E2 -27184.932} C_VEL
LIN {X 0,Y 171.206,Z 502.98,A -85,B 0,C 180,E1 -27188.335,E2 -27188.335} C_VEL
LIN {X 0,Y 171.747,Z 504.598,A -85,B 0,C 180,E1 -27189.273,E2 -27189.273} C_VEL
LIN {X 0,Y 169.191,Z 517.171,A -85,B 0,C 180,E1 -27189.895,E2 -27189.895} C_VEL
LIN {X 0,Y 165.366,Z 529.75,A -85,B 0,C 180,E1 -27190.728,E2 -27190.728} C_VEL
LIN {X 0,Y 160.658,Z 541.298,A -85,B 0,C 180,E1 -27191.826,E2 -27191.826} C_VEL
LIN {X 0,Y 154.726,Z 552.688,A -85,B 0,C 180,E1 -27193.274,E2 -27193.274} C_VEL
LIN {X 0,Y 148.234,Z 562.822,A -85,B 0,C 180,E1 -27194.987,E2 -27194.987} C_VEL
LIN {X 0,Y 141.439,Z 571.647,A -85,B 0,C 180,E1 -27196.962,E2 -27196.962} C_VEL
LIN {X 0,Y 134.11,Z 579.677,A -85,B 0,C 180,E1 -27199.393,E2 -27199.393} C_VEL
LIN {X 0,Y 125.899,Z 587.255,A -85,B 0,C 180,E1 -27202.587,E2 -27202.587} C_VEL
LIN {X 0,Y 117.7,Z 593.602,A -85,B 0,C 180,E1 -27206.408,E2 -27206.408} C_VEL
LIN {X 0,Y 110.344,Z 598.369,A -85,B 0,C 180,E1 -27210.634,E2 -27210.634} C_VEL
LIN {X 0,Y 103.525,Z 601.983,A -85,B 0,C 180,E1 -27215.45,E2 -27215.45} C_VEL
LIN {X 0,Y 98.421,Z 604.135,A -85,B 0,C 180,E1 -27219.993,E2 -27219.993} C_VEL
LIN {X 0,Y 92.575,Z 605.925,A -85,B 0,C 180,E1 -27226.903,E2 -27226.903} C_VEL
LIN {X 0,Y 89.616,Z 606.355,A -85,B 0,C 180,E1 -27231.652,E2 -27231.652} C_VEL
LIN {X 0,Y 85.786,Z 605.912,A -85,B 0,C 180,E1 -27240.558,E2 -27240.558} C_VEL
LIN {X 0,Y 84.434,Z 604.863,A -85,B 0,C 180,E1 -27246.295,E2 -27246.295} C_VEL
LIN {X 0,Y 83.651,Z 602.046,A -85,B 0,C 180,E1 -27255.402,E2 -27255.402} C_VEL
LIN {X 0,Y 84.352,Z 598.6,A -85,B 0,C 180,E1 -27262.823,E2 -27262.823} C_VEL
LIN {X 0,Y 86.018,Z 594.066,A -85,B 0,C 180,E1 -27270,E2 -27270} C_VEL
LIN {X 0,Y 88.575,Z 588.327,A -85,B 0,C 180,E1 -27276.835,E2 -27276.835} C_VEL
LIN {X 0,Y 92.119,Z 581.137,A -85,B 0,C 180,E1 -27283.231,E2 -27283.231} C_VEL
LIN {X 0,Y 96.52,Z 572.245,A -85,B 0,C 180,E1 -27289.076,E2 -27289.076} C_VEL
LIN {X 0,Y 100.915,Z 562.964,A -85,B 0,C 180,E1 -27293.605,E2 -27293.605} C_VEL
LIN {X 0,Y 104.678,Z 554.028,A -85,B 0,C 180,E1 -27296.948,E2 -27296.948} C_VEL
LIN {X 0,Y 108.774,Z 543.029,A -85,B 0,C 180,E1 -27300.048,E2 -27300.048} C_VEL
LIN {X 0,Y 112.59,Z 530.691,A -85,B 0,C 180,E1 -27302.573,E2 -27302.573} C_VEL
LIN {X 0,Y 115.602,Z 518.149,A -85,B 0,C 180,E1 -27304.393,E2 -27304.393} C_VEL
LIN {X 0,Y 117.727,Z 504.681,A -85,B 0,C 180,E1 -27305.71,E2 -27305.71} C_VEL
LIN {X 0,Y 119.664,Z 483.397,A -85,B 0,C 180,E1 -27306.828,E2 -27306.828} C_VEL
LIN {X 0,Y 121.31,Z 463.35,A -85,B 0,C 180,E1 -27307.746,E2 -27307.746} C_VEL
LIN {X 0,Y 116.937,Z 453.51,A -85,B 0,C 180,E1 -27311.011,E2 -27311.011} C_VEL
LIN {X 0,Y 112.909,Z 445.97,A -85,B 0,C 180,E1 -27314.317,E2 -27314.317} C_VEL
LIN {X 0,Y 108.901,Z 439.362,A -85,B 0,C 180,E1 -27318.052,E2 -27318.052} C_VEL
LIN {X 0,Y 106.217,Z 435.375,A -85,B 0,C 180,E1 -27320.899,E2 -27320.899} C_VEL
LIN {X 0,Y 104.057,Z 432.142,A -85,B 0,C 180,E1 -27323.492,E2 -27323.492} C_VEL
LIN {X 0,Y 101.524,Z 428.677,A -85,B 0,C 180,E1 -27326.943,E2 -27326.943} C_VEL
LIN {X 0,Y 100.933,Z 427.713,A -85,B 0,C 180,E1 -27327.869,E2 -27327.869} C_VEL
LIN {X 0,Y 98.072,Z 424.472,A -85,B 0,C 180,E1 -27332.815,E2 -27332.815} C_VEL
LIN {X 0,Y 97.185,Z 422.565,A -85,B 0,C 180,E1 -27334.929,E2 -27334.929} C_VEL
LIN {X 0,Y 94.013,Z 419.687,A -85,B 0,C 180,E1 -27345.69,E2 -27345.69} C_VEL
LIN {X 0,Y 93.721,Z 418.729,A -85,B 0,C 180,E1 -27349.194,E2 -27349.194} C_VEL
LIN {X 0,Y 93.677,Z 418.405,A -85,B 0,C 180,E1 -27351.369,E2 -27351.369} C_VEL
LIN {X 0,Y 94.44,Z 419.077,A -85,B 0,C 180,E1 -27359.466,E2 -27359.466} C_VEL
LIN {X 0,Y 95.917,Z 421.464,A -85,B 0,C 180,E1 -27365.254,E2 -27365.254} C_VEL
LIN {X 0,Y 97.702,Z 422.786,A -85,B 0,C 180,E1 -27369.444,E2 -27369.444} C_VEL
LIN {X 0,Y 99.416,Z 426.077,A -85,B 0,C 180,E1 -27373.022,E2 -27373.022} C_VEL
LIN {X 0,Y 101.533,Z 428.278,A -85,B 0,C 180,E1 -27376.328,E2 -27376.328} C_VEL
LIN {X 0,Y 103.853,Z 431.704,A -85,B 0,C 180,E1 -27379.571,E2 -27379.571} C_VEL
LIN {X 0,Y 104.895,Z 433.191,A -85,B 0,C 180,E1 -27380.866,E2 -27380.866} C_VEL
LIN {X 0,Y 107.719,Z 437.462,A -85,B 0,C 180,E1 -27384.054,E2 -27384.054} C_VEL
LIN {X 0,Y 111.632,Z 443.611,A -85,B 0,C 180,E1 -27387.856,E2 -27387.856} C_VEL
LIN {X 0,Y 114.762,Z 449.43,A -85,B 0,C 180,E1 -27390.585,E2 -27390.585} C_VEL
LIN {X 0,Y 118.01,Z 458.672,A -85,B 0,C 180,E1 -27393.412,E2 -27393.412} C_VEL
LIN {X 0,Y 120.293,Z 466.658,A -85,B 0,C 180,E1 -27395.351,E2 -27395.351} C_VEL
LIN {X 0,Y 120.467,Z 477.029,A -85,B 0,C 180,E1 -27396.341,E2 -27396.341} C_VEL
LIN {X 0,Y 117.584,Z 510.903,A -85,B 0,C 180,E1 -27398.004,E2 -27398.004} C_VEL
LIN {X 0,Y 115.339,Z 524.582,A -85,B 0,C 180,E1 -27399.197,E2 -27399.197} C_VEL
LIN {X 0,Y 112.541,Z 536.475,A -85,B 0,C 180,E1 -27400.785,E2 -27400.785} C_VEL
LIN {X 0,Y 109.62,Z 545.995,A -85,B 0,C 180,E1 -27402.5,E2 -27402.5} C_VEL
LIN {X 0,Y 105.668,Z 556.713,A -85,B 0,C 180,E1 -27405.036,E2 -27405.036} C_VEL
LIN {X 0,Y 102.535,Z 564.283,A -85,B 0,C 180,E1 -27407.403,E2 -27407.403} C_VEL
LIN {X 0,Y 98.291,Z 573.873,A -85,B 0,C 180,E1 -27411.273,E2 -27411.273} C_VEL
LIN {X 0,Y 94.945,Z 580.539,A -85,B 0,C 180,E1 -27414.693,E2 -27414.693} C_VEL
LIN {X 0,Y 91.182,Z 588.407,A -85,B 0,C 180,E1 -27419.935,E2 -27419.935} C_VEL
LIN {X 0,Y 87.777,Z 595.739,A -85,B 0,C 180,E1 -27426.402,E2 -27426.402} C_VEL
LIN {X 0,Y 85.466,Z 601.564,A -85,B 0,C 180,E1 -27433.273,E2 -27433.273} C_VEL
LIN {X 0,Y 84.362,Z 606.127,A -85,B 0,C 180,E1 -27440.409,E2 -27440.409} C_VEL
LIN {X 0,Y 84.147,Z 608.508,A -85,B 0,C 180,E1 -27445.209,E2 -27445.209} C_VEL
LIN {X 0,Y 84.275,Z 610.436,A -85,B 0,C 180,E1 -27450,E2 -27450} C_VEL
LIN {X 0,Y 84.137,Z 611.886,A -85,B 0,C 180,E1 -27454.791,E2 -27454.791} C_VEL
LIN {X 0,Y 85.008,Z 613.486,A -85,B 0,C 180,E1 -27464.36,E2 -27464.36} C_VEL
LIN {X 0,Y 87.967,Z 613.574,A -85,B 0,C 180,E1 -27473.544,E2 -27473.544} C_VEL
LIN {X 0,Y 90.368,Z 613.053,A -85,B 0,C 180,E1 -27477.815,E2 -27477.815} C_VEL
LIN {X 0,Y 96.548,Z 610.803,A -85,B 0,C 180,E1 -27485.615,E2 -27485.615} C_VEL
LIN {X 0,Y 102.584,Z 607.867,A -85,B 0,C 180,E1 -27491.097,E2 -27491.097} C_VEL
LIN {X 0,Y 110.941,Z 602.923,A -85,B 0,C 180,E1 -27496.76,E2 -27496.76} C_VEL
LIN {X 0,Y 119.538,Z 596.751,A -85,B 0,C 180,E1 -27501.168,E2 -27501.168} C_VEL
LIN {X 0,Y 127.484,Z 590.066,A -85,B 0,C 180,E1 -27504.402,E2 -27504.402} C_VEL
LIN {X 0,Y 135.856,Z 581.806,A -85,B 0,C 180,E1 -27507.205,E2 -27507.205} C_VEL
LIN {X 0,Y 143.058,Z 573.375,A -85,B 0,C 180,E1 -27509.283,E2 -27509.283} C_VEL
LIN {X 0,Y 150.506,Z 562.988,A -85,B 0,C 180,E1 -27511.108,E2 -27511.108} C_VEL
LIN {X 0,Y 157.358,Z 551.325,A -85,B 0,C 180,E1 -27512.579,E2 -27512.579} C_VEL
LIN {X 0,Y 162.736,Z 539.742,A -85,B 0,C 180,E1 -27513.65,E2 -27513.65} C_VEL
LIN {X 0,Y 167.177,Z 527.212,A -85,B 0,C 180,E1 -27514.467,E2 -27514.467} C_VEL
LIN {X 0,Y 170.525,Z 513.956,A -85,B 0,C 180,E1 -27515.051,E2 -27515.051} C_VEL
LIN {X 0,Y 171.368,Z 508.898,A -85,B 0,C 180,E1 -27515.27,E2 -27515.27} C_VEL
LIN {X 0,Y 169.743,Z 502.721,A -85,B 0,C 180,E1 -27518.282,E2 -27518.282} C_VEL
LIN {X 0,Y 168.111,Z 497.212,A -85,B 0,C 180,E1 -27521.885,E2 -27521.885} C_VEL
LIN {X 0,Y 167.366,Z 494.654,A -85,B 0,C 180,E1 -27524.046,E2 -27524.046} C_VEL
LIN {X 0,Y 167.031,Z 493.861,A -85,B 0,C 180,E1 -27525.109,E2 -27525.109} C_VEL
LIN {X 0,Y 166.448,Z 494.257,A -85,B 0,C 180,E1 -27526.672,E2 -27526.672} C_VEL
LIN {X 0,Y 165.317,Z 497.255,A -85,B 0,C 180,E1 -27530.329,E2 -27530.329} C_VEL
LIN {X 0,Y 165.203,Z 497.484,A -85,B 0,C 180,E1 -27531.287,E2 -27531.287} C_VEL
LIN {X 0,Y 165.344,Z 497.624,A -85,B 0,C 180,E1 -27534.971,E2 -27534.971} C_VEL
LIN {X 0,Y 166.27,Z 500.86,A -85,B 0,C 180,E1 -27540.001,E2 -27540.001} C_VEL
LIN {X 0,Y 167.635,Z 504.613,A -85,B 0,C 180,E1 -27543.907,E2 -27543.907} C_VEL
LIN {X 0,Y 168.903,Z 508.503,A -85,B 0,C 180,E1 -27546.898,E2 -27546.898} C_VEL
LIN {X 0,Y 169.032,Z 509.001,A -85,B 0,C 180,E1 -27547.203,E2 -27547.203} C_VEL
LIN {X 0,Y 165.959,Z 521.537,A -85,B 0,C 180,E1 -27547.826,E2 -27547.826} C_VEL
LIN {X 0,Y 161.722,Z 533.706,A -85,B 0,C 180,E1 -27548.648,E2 -27548.648} C_VEL
LIN {X 0,Y 156.29,Z 545.742,A -85,B 0,C 180,E1 -27549.867,E2 -27549.867} C_VEL
LIN {X 0,Y 149.655,Z 557.125,A -85,B 0,C 180,E1 -27551.392,E2 -27551.392} C_VEL
LIN {X 0,Y 142.558,Z 567.058,A -85,B 0,C 180,E1 -27553.185,E2 -27553.185} C_VEL
LIN {X 0,Y 135.538,Z 575.285,A -85,B 0,C 180,E1 -27555.195,E2 -27555.195} C_VEL
LIN {X 0,Y 127.353,Z 583.333,A -85,B 0,C 180,E1 -27557.84,E2 -27557.84} C_VEL
LIN {X 0,Y 118.719,Z 590.405,A -85,B 0,C 180,E1 -27561.195,E2 -27561.195} C_VEL
LIN {X 0,Y 109.231,Z 596.815,A -85,B 0,C 180,E1 -27565.744,E2 -27565.744} C_VEL
LIN {X 0,Y 101.724,Z 600.905,A -85,B 0,C 180,E1 -27570.278,E2 -27570.278} C_VEL
LIN {X 0,Y 93.02,Z 604.52,A -85,B 0,C 180,E1 -27577.189,E2 -27577.189} C_VEL
LIN {X 0,Y 87.245,Z 606.148,A -85,B 0,C 180,E1 -27583.533,E2 -27583.533} C_VEL
LIN {X 0,Y 83.316,Z 606.702,A -85,B 0,C 180,E1 -27589.395,E2 -27589.395} C_VEL
LIN {X 0,Y 79.392,Z 606.338,A -85,B 0,C 180,E1 -27597.918,E2 -27597.918} C_VEL
LIN {X 0,Y 77.48,Z 605.161,A -85,B 0,C 180,E1 -27605.108,E2 -27605.108} C_VEL
LIN {X 0,Y 76.55,Z 602.674,A -85,B 0,C 180,E1 -27614.013,E2 -27614.013} C_VEL
LIN {X 0,Y 77.12,Z 599.333,A -85,B 0,C 180,E1 -27622.144,E2 -27622.144} C_VEL
LIN {X 0,Y 78.784,Z 594.907,A -85,B 0,C 180,E1 -27630,E2 -27630} C_VEL
LIN {X 0,Y 81.431,Z 589.29,A -85,B 0,C 180,E1 -27637.438,E2 -27637.438} C_VEL
LIN {X 0,Y 85.171,Z 582.283,A -85,B 0,C 180,E1 -27644.332,E2 -27644.332} C_VEL
LIN {X 0,Y 89.836,Z 573.502,A -85,B 0,C 180,E1 -27650.614,E2 -27650.614} C_VEL
LIN {X 0,Y 94.409,Z 564.5,A -85,B 0,C 180,E1 -27655.343,E2 -27655.343} C_VEL
LIN {X 0,Y 98.895,Z 554.62,A -85,B 0,C 180,E1 -27659.246,E2 -27659.246} C_VEL
LIN {X 0,Y 103.221,Z 543.712,A -85,B 0,C 180,E1 -27662.424,E2 -27662.424} C_VEL
LIN {X 0,Y 107.222,Z 531.471,A -85,B 0,C 180,E1 -27664.996,E2 -27664.996} C_VEL
LIN {X 0,Y 110.535,Z 518.481,A -85,B 0,C 180,E1 -27666.904,E2 -27666.904} C_VEL
LIN {X 0,Y 112.716,Z 505.508,A -85,B 0,C 180,E1 -27668.191,E2 -27668.191} C_VEL
LIN {X 0,Y 114.621,Z 486.256,A -85,B 0,C 180,E1 -27669.222,E2 -27669.222} C_VEL
LIN {X 0,Y 116.387,Z 465.74,A -85,B 0,C 180,E1 -27670.163,E2 -27670.163} C_VEL
LIN {X 0,Y 112.685,Z 457.245,A -85,B 0,C 180,E1 -27673.275,E2 -27673.275} C_VEL
LIN {X 0,Y 109.147,Z 450.381,A -85,B 0,C 180,E1 -27676.545,E2 -27676.545} C_VEL
LIN {X 0,Y 105.738,Z 444.549,A -85,B 0,C 180,E1 -27680.109,E2 -27680.109} C_VEL
LIN {X 0,Y 103.313,Z 440.717,A -85,B 0,C 180,E1 -27682.999,E2 -27682.999} C_VEL
LIN {X 0,Y 101.719,Z 438.248,A -85,B 0,C 180,E1 -27685.121,E2 -27685.121} C_VEL
LIN {X 0,Y 98.856,Z 434.049,A -85,B 0,C 180,E1 -27689.545,E2 -27689.545} C_VEL
LIN {X 0,Y 96.209,Z 430.474,A -85,B 0,C 180,E1 -27694.806,E2 -27694.806} C_VEL
LIN {X 0,Y 95.767,Z 429.406,A -85,B 0,C 180,E1 -27696.015,E2 -27696.015} C_VEL
LIN {X 0,Y 92.979,Z 426.463,A -85,B 0,C 180,E1 -27706.892,E2 -27706.892} C_VEL
LIN {X 0,Y 92.789,Z 425.489,A -85,B 0,C 180,E1 -27711.286,E2 -27711.286} C_VEL
LIN {X 0,Y 93.393,Z 426.003,A -85,B 0,C 180,E1 -27718.651,E2 -27718.651} C_VEL
LIN {X 0,Y 95.013,Z 428.611,A -85,B 0,C 180,E1 -27725.304,E2 -27725.304} C_VEL
LIN {X 0,Y 96.148,Z 429.521,A -85,B 0,C 180,E1 -27728.141,E2 -27728.141} C_VEL
LIN {X 0,Y 97.947,Z 432.901,A -85,B 0,C 180,E1 -27732.167,E2 -27732.167} C_VEL
LIN {X 0,Y 99.589,Z 434.777,A -85,B 0,C 180,E1 -27734.952,E2 -27734.952} C_VEL
LIN {X 0,Y 102.614,Z 439.418,A -85,B 0,C 180,E1 -27739.408,E2 -27739.408} C_VEL
LIN {X 0,Y 105.757,Z 444.514,A -85,B 0,C 180,E1 -27743.239,E2 -27743.239} C_VEL
LIN {X 0,Y 108.973,Z 449.995,A -85,B 0,C 180,E1 -27746.603,E2 -27746.603} C_VEL
LIN {X 0,Y 111.135,Z 454.311,A -85,B 0,C 180,E1 -27748.683,E2 -27748.683} C_VEL
LIN {X 0,Y 114.025,Z 463.206,A -85,B 0,C 180,E1 -27751.512,E2 -27751.512} C_VEL
LIN {X 0,Y 115.518,Z 468.628,A -85,B 0,C 180,E1 -27752.936,E2 -27752.936} C_VEL
LIN {X 0,Y 115.621,Z 477.56,A -85,B 0,C 180,E1 -27753.843,E2 -27753.843} C_VEL
LIN {X 0,Y 112.626,Z 510.76,A -85,B 0,C 180,E1 -27755.479,E2 -27755.479} C_VEL
LIN {X 0,Y 110.32,Z 524.17,A -85,B 0,C 180,E1 -27756.652,E2 -27756.652} C_VEL
LIN {X 0,Y 107.378,Z 536.082,A -85,B 0,C 180,E1 -27758.243,E2 -27758.243} C_VEL
LIN {X 0,Y 104.322,Z 545.619,A -85,B 0,C 180,E1 -27759.978,E2 -27759.978} C_VEL
LIN {X 0,Y 100.165,Z 556.347,A -85,B 0,C 180,E1 -27762.548,E2 -27762.548} C_VEL
LIN {X 0,Y 96.847,Z 563.921,A -85,B 0,C 180,E1 -27764.967,E2 -27764.967} C_VEL
LIN {X 0,Y 92.179,Z 573.809,A -85,B 0,C 180,E1 -27769.102,E2 -27769.102} C_VEL
LIN {X 0,Y 88.718,Z 580.289,A -85,B 0,C 180,E1 -27772.596,E2 -27772.596} C_VEL
LIN {X 0,Y 85.068,Z 587.371,A -85,B 0,C 180,E1 -27777.521,E2 -27777.521} C_VEL
LIN {X 0,Y 81.283,Z 594.828,A -85,B 0,C 180,E1 -27784.386,E2 -27784.386} C_VEL
LIN {X 0,Y 78.664,Z 600.782,A -85,B 0,C 180,E1 -27791.779,E2 -27791.779} C_VEL
LIN {X 0,Y 77.346,Z 605.454,A -85,B 0,C 180,E1 -27799.53,E2 -27799.53} C_VEL
LIN {X 0,Y 77.067,Z 607.9,A -85,B 0,C 180,E1 -27804.768,E2 -27804.768} C_VEL
LIN {X 0,Y 77.189,Z 609.874,A -85,B 0,C 180,E1 -27810,E2 -27810} C_VEL
LIN {X 0,Y 77.056,Z 611.368,A -85,B 0,C 180,E1 -27815.233,E2 -27815.233} C_VEL
LIN {X 0,Y 77.312,Z 612.441,A -85,B 0,C 180,E1 -27820.475,E2 -27820.475} C_VEL
LIN {X 0,Y 79.517,Z 613.359,A -85,B 0,C 180,E1 -27830.703,E2 -27830.703} C_VEL
LIN {X 0,Y 84.128,Z 612.794,A -85,B 0,C 180,E1 -27840.081,E2 -27840.081} C_VEL
LIN {X 0,Y 87.245,Z 611.926,A -85,B 0,C 180,E1 -27844.324,E2 -27844.324} C_VEL
LIN {X 0,Y 94.814,Z 608.991,A -85,B 0,C 180,E1 -27851.844,E2 -27851.844} C_VEL
LIN {X 0,Y 101.403,Z 605.702,A -85,B 0,C 180,E1 -27856.695,E2 -27856.695} C_VEL
LIN {X 0,Y 108.701,Z 601.385,A -85,B 0,C 180,E1 -27860.881,E2 -27860.881} C_VEL
LIN {X 0,Y 117.938,Z 594.909,A -85,B 0,C 180,E1 -27865.02,E2 -27865.02} C_VEL
LIN {X 0,Y 126.331,Z 587.865,A -85,B 0,C 180,E1 -27868.034,E2 -27868.034} C_VEL
LIN {X 0,Y 135.121,Z 579.097,A -85,B 0,C 180,E1 -27870.598,E2 -27870.598} C_VEL
LIN {X 0,Y 143.357,Z 569.187,A -85,B 0,C 180,E1 -27872.692,E2 -27872.692} C_VEL
LIN {X 0,Y 150.315,Z 559.117,A -85,B 0,C 180,E1 -27874.16,E2 -27874.16} C_VEL
LIN {X 0,Y 156.587,Z 547.973,A -85,B 0,C 180,E1 -27875.347,E2 -27875.347} C_VEL
LIN {X 0,Y 161.814,Z 536.26,A -85,B 0,C 180,E1 -27876.267,E2 -27876.267} C_VEL
LIN {X 0,Y 166.192,Z 523.163,A -85,B 0,C 180,E1 -27876.989,E2 -27876.989} C_VEL
LIN {X 0,Y 168.679,Z 512.459,A -85,B 0,C 180,E1 -27877.449,E2 -27877.449} C_VEL
LIN {X 0,Y 167.63,Z 507.19,A -85,B 0,C 180,E1 -27880.324,E2 -27880.324} C_VEL
LIN {X 0,Y 166.693,Z 503.441,A -85,B 0,C 180,E1 -27882.993,E2 -27882.993} C_VEL
LIN {X 0,Y 166.021,Z 500.707,A -85,B 0,C 180,E1 -27885.497,E2 -27885.497} C_VEL
LIN {X 0,Y 165.236,Z 497.499,A -85,B 0,C 180,E1 -27890.823,E2 -27890.823} C_VEL
LIN {X 0,Y 165.203,Z 497.484,A -85,B 0,C 180,E1 -27891.287,E2 -27891.287} C_VEL
LIN {X 0,Y 165.126,Z 497.855,A -85,B 0,C 180,E1 -27892.639,E2 -27892.639} C_VEL
LIN {X 0,Y 165.044,Z 499.612,A -85,B 0,C 180,E1 -27894.597,E2 -27894.597} C_VEL
LIN {X 0,Y 164.975,Z 502.233,A -85,B 0,C 180,E1 -27896.457,E2 -27896.457} C_VEL
LIN {X 0,Y 165.112,Z 508.019,A -85,B 0,C 180,E1 -27900.19,E2 -27900.19} C_VEL
LIN {X 0,Y 165.382,Z 509.481,A -85,B 0,C 180,E1 -27901.498,E2 -27901.498} C_VEL
LIN {X 0,Y 166.157,Z 512.362,A -85,B 0,C 180,E1 -27904.246,E2 -27904.246} C_VEL
LIN {X 0,Y 166.389,Z 513.334,A -85,B 0,C 180,E1 -27904.998,E2 -27904.998} C_VEL
LIN {X 0,Y 162.995,Z 525.528,A -85,B 0,C 180,E1 -27905.653,E2 -27905.653} C_VEL
LIN {X 0,Y 158.273,Z 537.647,A -85,B 0,C 180,E1 -27906.524,E2 -27906.524} C_VEL
LIN {X 0,Y 152.911,Z 548.434,A -85,B 0,C 180,E1 -27907.636,E2 -27907.636} C_VEL
LIN {X 0,Y 145.917,Z 559.662,A -85,B 0,C 180,E1 -27909.124,E2 -27909.124} C_VEL
LIN {X 0,Y 139.438,Z 568.192,A -85,B 0,C 180,E1 -27910.636,E2 -27910.636} C_VEL
LIN {X 0,Y 131.761,Z 576.71,A -85,B 0,C 180,E1 -27912.67,E2 -27912.67} C_VEL
LIN {X 0,Y 123.738,Z 584.165,A -85,B 0,C 180,E1 -27915.087,E2 -27915.087} C_VEL
LIN {X 0,Y 114.373,Z 591.419,A -85,B 0,C 180,E1 -27918.49,E2 -27918.49} C_VEL
LIN {X 0,Y 106.191,Z 596.648,A -85,B 0,C 180,E1 -27922.099,E2 -27922.099} C_VEL
LIN {X 0,Y 98.171,Z 600.869,A -85,B 0,C 180,E1 -27926.511,E2 -27926.511} C_VEL
LIN {X 0,Y 90.777,Z 603.935,A -85,B 0,C 180,E1 -27931.614,E2 -27931.614} C_VEL
LIN {X 0,Y 86.292,Z 605.385,A -85,B 0,C 180,E1 -27935.47,E2 -27935.47} C_VEL
LIN {X 0,Y 82.247,Z 606.371,A -85,B 0,C 180,E1 -27939.733,E2 -27939.733} C_VEL
LIN {X 0,Y 77.197,Z 607.047,A -85,B 0,C 180,E1 -27946.748,E2 -27946.748} C_VEL
LIN {X 0,Y 73.172,Z 606.766,A -85,B 0,C 180,E1 -27954.811,E2 -27954.811} C_VEL
LIN {X 0,Y 70.583,Z 605.465,A -85,B 0,C 180,E1 -27963.659,E2 -27963.659} C_VEL
LIN {X 0,Y 69.474,Z 602.355,A -85,B 0,C 180,E1 -27975.351,E2 -27975.351} C_VEL
LIN {X 0,Y 70.503,Z 598.177,A -85,B 0,C 180,E1 -27985.468,E2 -27985.468} C_VEL
LIN {X 0,Y 72.358,Z 594.078,A -85,B 0,C 180,E1 -27992.784,E2 -27992.784} C_VEL
LIN {X 0,Y 76.126,Z 587.003,A -85,B 0,C 180,E1 -28001.989,E2 -28001.989} C_VEL
LIN {X 0,Y 80.581,Z 579.355,A -85,B 0,C 180,E1 -28009.09,E2 -28009.09} C_VEL
LIN {X 0,Y 85.597,Z 570.434,A -85,B 0,C 180,E1 -28015.052,E2 -28015.052} C_VEL
LIN {X 0,Y 90.523,Z 560.935,A -85,B 0,C 180,E1 -28019.665,E2 -28019.665} C_VEL
LIN {X 0,Y 95.532,Z 550.11,A -85,B 0,C 180,E1 -28023.487,E2 -28023.487} C_VEL
LIN {X 0,Y 99.654,Z 539.599,A -85,B 0,C 180,E1 -28026.201,E2 -28026.201} C_VEL
LIN {X 0,Y 103.621,Z 526.971,A -85,B 0,C 180,E1 -28028.541,E2 -28028.541} C_VEL
LIN {X 0,Y 106.553,Z 514.461,A -85,B 0,C 180,E1 -28030.163,E2 -28030.163} C_VEL
LIN {X 0,Y 108.609,Z 501.197,A -85,B 0,C 180,E1 -28031.256,E2 -28031.256} C_VEL
LIN {X 0,Y 111.614,Z 468.072,A -85,B 0,C 180,E1 -28032.847,E2 -28032.847} C_VEL
LIN {X 0,Y 108.148,Z 459.959,A -85,B 0,C 180,E1 -28036.191,E2 -28036.191} C_VEL
LIN {X 0,Y 104.402,Z 452.622,A -85,B 0,C 180,E1 -28040.252,E2 -28040.252} C_VEL
LIN {X 0,Y 101.277,Z 447.276,A -85,B 0,C 180,E1 -28044.19,E2 -28044.19} C_VEL
LIN {X 0,Y 99.34,Z 444.164,A -85,B 0,C 180,E1 -28047.011,E2 -28047.011} C_VEL
LIN {X 0,Y 97.014,Z 440.499,A -85,B 0,C 180,E1 -28051.021,E2 -28051.021} C_VEL
LIN {X 0,Y 94.546,Z 436.675,A -85,B 0,C 180,E1 -28056.626,E2 -28056.626} C_VEL
LIN {X 0,Y 94.038,Z 436.046,A -85,B 0,C 180,E1 -28058.056,E2 -28058.056} C_VEL
LIN {X 0,Y 91.901,Z 432.574,A -85,B 0,C 180,E1 -28071.201,E2 -28071.201} C_VEL
LIN {X 0,Y 92.368,Z 432.911,A -85,B 0,C 180,E1 -28077.819,E2 -28077.819} C_VEL
LIN {X 0,Y 93.756,Z 435.398,A -85,B 0,C 180,E1 -28084.298,E2 -28084.298} C_VEL
LIN {X 0,Y 94.693,Z 436.319,A -85,B 0,C 180,E1 -28086.926,E2 -28086.926} C_VEL
LIN {X 0,Y 96.759,Z 440.028,A -85,B 0,C 180,E1 -28091.787,E2 -28091.787} C_VEL
LIN {X 0,Y 97.772,Z 441.372,A -85,B 0,C 180,E1 -28093.642,E2 -28093.642} C_VEL
LIN {X 0,Y 100.337,Z 445.54,A -85,B 0,C 180,E1 -28097.788,E2 -28097.788} C_VEL
LIN {X 0,Y 103.881,Z 451.536,A -85,B 0,C 180,E1 -28102.449,E2 -28102.449} C_VEL
LIN {X 0,Y 107.455,Z 458.625,A -85,B 0,C 180,E1 -28106.442,E2 -28106.442} C_VEL
LIN {X 0,Y 110.027,Z 467.316,A -85,B 0,C 180,E1 -28109.33,E2 -28109.33} C_VEL
LIN {X 0,Y 111.039,Z 471.737,A -85,B 0,C 180,E1 -28110.486,E2 -28110.486} C_VEL
LIN {X 0,Y 110.878,Z 479.593,A -85,B 0,C 180,E1 -28111.201,E2 -28111.201} C_VEL
LIN {X 0,Y 107.979,Z 510.095,A -85,B 0,C 180,E1 -28112.69,E2 -28112.69} C_VEL
LIN {X 0,Y 105.506,Z 523.897,A -85,B 0,C 180,E1 -28113.884,E2 -28113.884} C_VEL
LIN {X 0,Y 102.122,Z 536.731,A -85,B 0,C 180,E1 -28115.619,E2 -28115.619} C_VEL
LIN {X 0,Y 98.65,Z 546.961,A -85,B 0,C 180,E1 -28117.576,E2 -28117.576} C_VEL
LIN {X 0,Y 93.597,Z 558.58,A -85,B 0,C 180,E1 -28120.514,E2 -28120.514} C_VEL
LIN {X 0,Y 88.563,Z 569.127,A -85,B 0,C 180,E1 -28124.423,E2 -28124.423} C_VEL
LIN {X 0,Y 84.276,Z 577.395,A -85,B 0,C 180,E1 -28128.635,E2 -28128.635} C_VEL
LIN {X 0,Y 80.664,Z 583.369,A -85,B 0,C 180,E1 -28132.42,E2 -28132.42} C_VEL
LIN {X 0,Y 76.207,Z 591.588,A -85,B 0,C 180,E1 -28139.522,E2 -28139.522} C_VEL
LIN {X 0,Y 72.732,Z 598.132,A -85,B 0,C 180,E1 -28147.263,E2 -28147.263} C_VEL
LIN {X 0,Y 70.72,Z 603.311,A -85,B 0,C 180,E1 -28155.615,E2 -28155.615} C_VEL
LIN {X 0,Y 69.991,Z 607.293,A -85,B 0,C 180,E1 -28164.237,E2 -28164.237} C_VEL
LIN {X 0,Y 70.088,Z 609.311,A -85,B 0,C 180,E1 -28170,E2 -28170} C_VEL
LIN {X 0,Y 70.003,Z 610.848,A -85,B 0,C 180,E1 -28175.762,E2 -28175.762} C_VEL
LIN {X 0,Y 70.319,Z 611.973,A -85,B 0,C 180,E1 -28181.53,E2 -28181.53} C_VEL
LIN {X 0,Y 71.304,Z 612.692,A -85,B 0,C 180,E1 -28187.199,E2 -28187.199} C_VEL
LIN {X 0,Y 75.109,Z 612.943,A -85,B 0,C 180,E1 -28197.894,E2 -28197.894} C_VEL
LIN {X 0,Y 81.455,Z 611.722,A -85,B 0,C 180,E1 -28207.153,E2 -28207.153} C_VEL
LIN {X 0,Y 85.388,Z 610.505,A -85,B 0,C 180,E1 -28211.181,E2 -28211.181} C_VEL
LIN {X 0,Y 94.219,Z 606.863,A -85,B 0,C 180,E1 -28218.237,E2 -28218.237} C_VEL
LIN {X 0,Y 101.728,Z 602.988,A -85,B 0,C 180,E1 -28222.605,E2 -28222.605} C_VEL
LIN {X 0,Y 109.804,Z 598.024,A -85,B 0,C 180,E1 -28226.309,E2 -28226.309} C_VEL
LIN {X 0,Y 118.338,Z 591.821,A -85,B 0,C 180,E1 -28229.443,E2 -28229.443} C_VEL
LIN {X 0,Y 127.214,Z 584.139,A -85,B 0,C 180,E1 -28232.117,E2 -28232.117} C_VEL
LIN {X 0,Y 136.393,Z 574.53,A -85,B 0,C 180,E1 -28234.384,E2 -28234.384} C_VEL
LIN {X 0,Y 144.214,Z 564.656,A -85,B 0,C 180,E1 -28236.025,E2 -28236.025} C_VEL
LIN {X 0,Y 151.384,Z 553.585,A -85,B 0,C 180,E1 -28237.321,E2 -28237.321} C_VEL
LIN {X 0,Y 157.802,Z 541.043,A -85,B 0,C 180,E1 -28238.385,E2 -28238.385} C_VEL
LIN {X 0,Y 162.281,Z 529.763,A -85,B 0,C 180,E1 -28239.05,E2 -28239.05} C_VEL
LIN {X 0,Y 165.822,Z 517.669,A -85,B 0,C 180,E1 -28239.556,E2 -28239.556} C_VEL
LIN {X 0,Y 166.109,Z 516.207,A -85,B 0,C 180,E1 -28239.667,E2 -28239.667} C_VEL
LIN {X 0,Y 165.466,Z 511.604,A -85,B 0,C 180,E1 -28242.545,E2 -28242.545} C_VEL
LIN {X 0,Y 164.819,Z 507.682,A -85,B 0,C 180,E1 -28245.808,E2 -28245.808} C_VEL
LIN {X 0,Y 164.218,Z 504.512,A -85,B 0,C 180,E1 -28251.386,E2 -28251.386} C_VEL
LIN {X 0,Y 164.303,Z 504.658,A -85,B 0,C 180,E1 -28254.632,E2 -28254.632} C_VEL
LIN {X 0,Y 165.088,Z 508.333,A -85,B 0,C 180,E1 -28260.305,E2 -28260.305} C_VEL
LIN {X 0,Y 165.382,Z 509.481,A -85,B 0,C 180,E1 -28261.498,E2 -28261.498} C_VEL
LIN {X 0,Y 165.407,Z 511.036,A -85,B 0,C 180,E1 -28262.286,E2 -28262.286} C_VEL
LIN {X 0,Y 164.991,Z 514.022,A -85,B 0,C 180,E1 -28262.911,E2 -28262.911} C_VEL
LIN {X 0,Y 164.1,Z 517.78,A -85,B 0,C 180,E1 -28263.223,E2 -28263.223} C_VEL
LIN {X 0,Y 161.198,Z 526.62,A -85,B 0,C 180,E1 -28263.302,E2 -28263.302} C_VEL
LIN {X 0,Y 160.155,Z 529.401,A -85,B 0,C 180,E1 -28263.412,E2 -28263.412} C_VEL
LIN {X 0,Y 155.049,Z 541.372,A -85,B 0,C 180,E1 -28264.301,E2 -28264.301} C_VEL
LIN {X 0,Y 149.216,Z 552.033,A -85,B 0,C 180,E1 -28265.406,E2 -28265.406} C_VEL
LIN {X 0,Y 142.422,Z 562.079,A -85,B 0,C 180,E1 -28266.748,E2 -28266.748} C_VEL
LIN {X 0,Y 134.962,Z 571.184,A -85,B 0,C 180,E1 -28268.358,E2 -28268.358} C_VEL
LIN {X 0,Y 126.815,Z 579.483,A -85,B 0,C 180,E1 -28270.37,E2 -28270.37} C_VEL
LIN {X 0,Y 118.855,Z 586.297,A -85,B 0,C 180,E1 -28272.674,E2 -28272.674} C_VEL
LIN {X 0,Y 109.576,Z 592.912,A -85,B 0,C 180,E1 -28275.836,E2 -28275.836} C_VEL
LIN {X 0,Y 100.702,Z 598.071,A -85,B 0,C 180,E1 -28279.586,E2 -28279.586} C_VEL
LIN {X 0,Y 92.323,Z 602.006,A -85,B 0,C 180,E1 -28284.011,E2 -28284.011} C_VEL
LIN {X 0,Y 83.018,Z 605.291,A -85,B 0,C 180,E1 -28290.528,E2 -28290.528} C_VEL
LIN {X 0,Y 77.66,Z 606.594,A -85,B 0,C 180,E1 -28295.467,E2 -28295.467} C_VEL
LIN {X 0,Y 71.258,Z 607.393,A -85,B 0,C 180,E1 -28303.664,E2 -28303.664} C_VEL
LIN {X 0,Y 67.204,Z 607.193,A -85,B 0,C 180,E1 -28311.138,E2 -28311.138} C_VEL
LIN {X 0,Y 63.758,Z 605.774,A -85,B 0,C 180,E1 -28321.868,E2 -28321.868} C_VEL
LIN {X 0,Y 62.534,Z 603.929,A -85,B 0,C 180,E1 -28330.296,E2 -28330.296} C_VEL
LIN {X 0,Y 62.659,Z 600.8,A -85,B 0,C 180,E1 -28340.314,E2 -28340.314} C_VEL
LIN {X 0,Y 64.306,Z 596.592,A -85,B 0,C 180,E1 -28350,E2 -28350} C_VEL
LIN {X 0,Y 67.804,Z 590.183,A -85,B 0,C 180,E1 -28360.451,E2 -28360.451} C_VEL
LIN {X 0,Y 72.16,Z 583.225,A -85,B 0,C 180,E1 -28368.453,E2 -28368.453} C_VEL
LIN {X 0,Y 76.591,Z 576.132,A -85,B 0,C 180,E1 -28374.388,E2 -28374.388} C_VEL
LIN {X 0,Y 81.876,Z 567.264,A -85,B 0,C 180,E1 -28379.797,E2 -28379.797} C_VEL
LIN {X 0,Y 87.236,Z 557.012,A -85,B 0,C 180,E1 -28384.328,E2 -28384.328} C_VEL
LIN {X 0,Y 92.147,Z 546.499,A -85,B 0,C 180,E1 -28387.6,E2 -28387.6} C_VEL
LIN {X 0,Y 96.548,Z 534.991,A -85,B 0,C 180,E1 -28390.242,E2 -28390.242} C_VEL
LIN {X 0,Y 100.133,Z 523.068,A -85,B 0,C 180,E1 -28392.156,E2 -28392.156} C_VEL
LIN {X 0,Y 102.949,Z 509.996,A -85,B 0,C 180,E1 -28393.606,E2 -28393.606} C_VEL
LIN {X 0,Y 104.757,Z 496.476,A -85,B 0,C 180,E1 -28394.497,E2 -28394.497} C_VEL
LIN {X 0,Y 107.189,Z 470.66,A -85,B 0,C 180,E1 -28395.672,E2 -28395.672} C_VEL
LIN {X 0,Y 103.682,Z 462.369,A -85,B 0,C 180,E1 -28399.602,E2 -28399.602} C_VEL
LIN {X 0,Y 100.578,Z 456.198,A -85,B 0,C 180,E1 -28403.573,E2 -28403.573} C_VEL
LIN {X 0,Y 97.492,Z 450.685,A -85,B 0,C 180,E1 -28408.277,E2 -28408.277} C_VEL
LIN {X 0,Y 95.247,Z 446.941,A -85,B 0,C 180,E1 -28412.535,E2 -28412.535} C_VEL
LIN {X 0,Y 93.007,Z 443.055,A -85,B 0,C 180,E1 -28418.383,E2 -28418.383} C_VEL
LIN {X 0,Y 91.014,Z 439.655,A -85,B 0,C 180,E1 -28431.115,E2 -28431.115} C_VEL
LIN {X 0,Y 91.323,Z 439.826,A -85,B 0,C 180,E1 -28436.691,E2 -28436.691} C_VEL
LIN {X 0,Y 93.328,Z 443.17,A -85,B 0,C 180,E1 -28445.807,E2 -28445.807} C_VEL
LIN {X 0,Y 95.197,Z 446.679,A -85,B 0,C 180,E1 -28450.635,E2 -28450.635} C_VEL
LIN {X 0,Y 96.068,Z 448.059,A -85,B 0,C 180,E1 -28452.409,E2 -28452.409} C_VEL
LIN {X 0,Y 98.226,Z 451.763,A -85,B 0,C 180,E1 -28456.229,E2 -28456.229} C_VEL
LIN {X 0,Y 101.505,Z 457.837,A -85,B 0,C 180,E1 -28460.999,E2 -28460.999} C_VEL
LIN {X 0,Y 104.167,Z 463.599,A -85,B 0,C 180,E1 -28464.325,E2 -28464.325} C_VEL
LIN {X 0,Y 106.609,Z 472.919,A -85,B 0,C 180,E1 -28467.481,E2 -28467.481} C_VEL
LIN {X 0,Y 106.669,Z 478.721,A -85,B 0,C 180,E1 -28468.201,E2 -28468.201} C_VEL
LIN {X 0,Y 103.517,Z 510.045,A -85,B 0,C 180,E1 -28469.699,E2 -28469.699} C_VEL
LIN {X 0,Y 100.956,Z 523.646,A -85,B 0,C 180,E1 -28470.86,E2 -28470.86} C_VEL
LIN {X 0,Y 97.452,Z 536.349,A -85,B 0,C 180,E1 -28472.558,E2 -28472.558} C_VEL
LIN {X 0,Y 93.798,Z 546.589,A -85,B 0,C 180,E1 -28474.495,E2 -28474.495} C_VEL
LIN {X 0,Y 88.501,Z 558.22,A -85,B 0,C 180,E1 -28477.43,E2 -28477.43} C_VEL
LIN {X 0,Y 83.126,Z 568.767,A -85,B 0,C 180,E1 -28481.381,E2 -28481.381} C_VEL
LIN {X 0,Y 77.754,Z 578.219,A -85,B 0,C 180,E1 -28486.415,E2 -28486.415} C_VEL
LIN {X 0,Y 74.214,Z 583.781,A -85,B 0,C 180,E1 -28490.267,E2 -28490.267} C_VEL
LIN {X 0,Y 69.413,Z 591.863,A -85,B 0,C 180,E1 -28497.89,E2 -28497.89} C_VEL
LIN {X 0,Y 66.193,Z 597.282,A -85,B 0,C 180,E1 -28504.869,E2 -28504.869} C_VEL
LIN {X 0,Y 63.816,Z 602.583,A -85,B 0,C 180,E1 -28514.019,E2 -28514.019} C_VEL
LIN {X 0,Y 62.917,Z 606.663,A -85,B 0,C 180,E1 -28523.587,E2 -28523.587} C_VEL
LIN {X 0,Y 62.999,Z 608.749,A -85,B 0,C 180,E1 -28530,E2 -28530} C_VEL
LIN {X 0,Y 62.946,Z 610.328,A -85,B 0,C 180,E1 -28536.41,E2 -28536.41} C_VEL
LIN {X 0,Y 64.52,Z 612.276,A -85,B 0,C 180,E1 -28549.073,E2 -28549.073} C_VEL
LIN {X 0,Y 68.892,Z 612.628,A -85,B 0,C 180,E1 -28560.668,E2 -28560.668} C_VEL
LIN {X 0,Y 75.898,Z 611.492,A -85,B 0,C 180,E1 -28570.404,E2 -28570.404} C_VEL
LIN {X 0,Y 80.158,Z 610.353,A -85,B 0,C 180,E1 -28574.539,E2 -28574.539} C_VEL
LIN {X 0,Y 89.643,Z 606.802,A -85,B 0,C 180,E1 -28581.626,E2 -28581.626} C_VEL
LIN {X 0,Y 97.579,Z 603.018,A -85,B 0,C 180,E1 -28585.92,E2 -28585.92} C_VEL
LIN {X 0,Y 106.036,Z 598.153,A -85,B 0,C 180,E1 -28589.498,E2 -28589.498} C_VEL
LIN {X 0,Y 116.41,Z 590.949,A -85,B 0,C 180,E1 -28592.934,E2 -28592.934} C_VEL
LIN {X 0,Y 125.634,Z 583.11,A -85,B 0,C 180,E1 -28595.369,E2 -28595.369} C_VEL
LIN {X 0,Y 135.081,Z 573.382,A -85,B 0,C 180,E1 -28597.44,E2 -28597.44} C_VEL
LIN {X 0,Y 143.109,Z 563.324,A -85,B 0,C 180,E1 -28598.917,E2 -28598.917} C_VEL
LIN {X 0,Y 150.438,Z 551.966,A -85,B 0,C 180,E1 -28600.077,E2 -28600.077} C_VEL
LIN {X 0,Y 156.172,Z 540.867,A -85,B 0,C 180,E1 -28600.911,E2 -28600.911} C_VEL
LIN {X 0,Y 160.96,Z 528.985,A -85,B 0,C 180,E1 -28601.547,E2 -28601.547} C_VEL
LIN {X 0,Y 163.603,Z 520.366,A -85,B 0,C 180,E1 -28601.873,E2 -28601.873} C_VEL
LIN {X 0,Y 163.382,Z 516.662,A -85,B 0,C 180,E1 -28604.405,E2 -28604.405} C_VEL
LIN {X 0,Y 163.159,Z 514.229,A -85,B 0,C 180,E1 -28606.614,E2 -28606.614} C_VEL
LIN {X 0,Y 162.886,Z 511.559,A -85,B 0,C 180,E1 -28611.315,E2 -28611.315} C_VEL
LIN {X 0,Y 162.907,Z 511.567,A -85,B 0,C 180,E1 -28614.274,E2 -28614.274} C_VEL
LIN {X 0,Y 163.333,Z 515.119,A -85,B 0,C 180,E1 -28619.847,E2 -28619.847} C_VEL
LIN {X 0,Y 163.809,Z 517.95,A -85,B 0,C 180,E1 -28622.767,E2 -28622.767} C_VEL
LIN {X 0,Y 160.155,Z 529.401,A -85,B 0,C 180,E1 -28623.412,E2 -28623.412} C_VEL
LIN {X 0,Y 157.911,Z 534.866,A -85,B 0,C 180,E1 -28623.548,E2 -28623.548} C_VEL
LIN {X 0,Y 153.352,Z 543.638,A -85,B 0,C 180,E1 -28623.21,E2 -28623.21} C_VEL
LIN {X 0,Y 148.112,Z 552.005,A -85,B 0,C 180,E1 -28622.936,E2 -28622.936} C_VEL
LIN {X 0,Y 144.794,Z 556.83,A -85,B 0,C 180,E1 -28623.21,E2 -28623.21} C_VEL
LIN {X 0,Y 136.625,Z 567.538,A -85,B 0,C 180,E1 -28624.704,E2 -28624.704} C_VEL
LIN {X 0,Y 127.359,Z 577.396,A -85,B 0,C 180,E1 -28626.656,E2 -28626.656} C_VEL
LIN {X 0,Y 117.439,Z 585.896,A -85,B 0,C 180,E1 -28629.106,E2 -28629.106} C_VEL
LIN {X 0,Y 107.781,Z 592.671,A -85,B 0,C 180,E1 -28632.021,E2 -28632.021} C_VEL
LIN {X 0,Y 98.452,Z 597.983,A -85,B 0,C 180,E1 -28635.49,E2 -28635.49} C_VEL
LIN {X 0,Y 89.54,Z 602.026,A -85,B 0,C 180,E1 -28639.635,E2 -28639.635} C_VEL
LIN {X 0,Y 83.899,Z 604.069,A -85,B 0,C 180,E1 -28642.866,E2 -28642.866} C_VEL
LIN {X 0,Y 78.487,Z 605.687,A -85,B 0,C 180,E1 -28646.599,E2 -28646.599} C_VEL
LIN {X 0,Y 73.568,Z 606.816,A -85,B 0,C 180,E1 -28650.711,E2 -28650.711} C_VEL
LIN {X 0,Y 65.571,Z 607.738,A -85,B 0,C 180,E1 -28660.025,E2 -28660.025} C_VEL
LIN {X 0,Y 61.575,Z 607.608,A -85,B 0,C 180,E1 -28666.78,E2 -28666.78} C_VEL
LIN {X 0,Y 57.019,Z 606.086,A -85,B 0,C 180,E1 -28679.637,E2 -28679.637} C_VEL
LIN {X 0,Y 55.64,Z 604.524,A -85,B 0,C 180,E1 -28687.733,E2 -28687.733} C_VEL
LIN {X 0,Y 55.457,Z 601.496,A -85,B 0,C 180,E1 -28699.042,E2 -28699.042} C_VEL
LIN {X 0,Y 57.027,Z 597.409,A -85,B 0,C 180,E1 -28710,E2 -28710} C_VEL
LIN {X 0,Y 60.762,Z 591.142,A -85,B 0,C 180,E1 -28721.678,E2 -28721.678} C_VEL
LIN {X 0,Y 65.364,Z 584.327,A -85,B 0,C 180,E1 -28730.453,E2 -28730.453} C_VEL
LIN {X 0,Y 71.17,Z 575.867,A -85,B 0,C 180,E1 -28737.972,E2 -28737.972} C_VEL
LIN {X 0,Y 76.748,Z 567.133,A -85,B 0,C 180,E1 -28743.327,E2 -28743.327} C_VEL
LIN {X 0,Y 82.063,Z 557.604,A -85,B 0,C 180,E1 -28747.602,E2 -28747.602} C_VEL
LIN {X 0,Y 87.256,Z 547.149,A -85,B 0,C 180,E1 -28750.875,E2 -28750.875} C_VEL
LIN {X 0,Y 91.895,Z 535.732,A -85,B 0,C 180,E1 -28753.495,E2 -28753.495} C_VEL
LIN {X 0,Y 95.67,Z 523.974,A -85,B 0,C 180,E1 -28755.368,E2 -28755.368} C_VEL
LIN {X 0,Y 98.681,Z 510.893,A -85,B 0,C 180,E1 -28756.802,E2 -28756.802} C_VEL
LIN {X 0,Y 100.48,Z 498.556,A -85,B 0,C 180,E1 -28757.647,E2 -28757.647} C_VEL
LIN {X 0,Y 102.961,Z 473.283,A -85,B 0,C 180,E1 -28758.803,E2 -28758.803} C_VEL
LIN {X 0,Y 100.314,Z 466.729,A -85,B 0,C 180,E1 -28762.261,E2 -28762.261} C_VEL
LIN {X 0,Y 97.757,Z 461.254,A -85,B 0,C 180,E1 -28766.03,E2 -28766.03} C_VEL
LIN {X 0,Y 95.254,Z 456.536,A -85,B 0,C 180,E1 -28770.393,E2 -28770.393} C_VEL
LIN {X 0,Y 93.522,Z 453.341,A -85,B 0,C 180,E1 -28774.168,E2 -28774.168} C_VEL
LIN {X 0,Y 91.633,Z 449.827,A -85,B 0,C 180,E1 -28779.808,E2 -28779.808} C_VEL
LIN {X 0,Y 90.126,Z 446.743,A -85,B 0,C 180,E1 -28791.026,E2 -28791.026} C_VEL
LIN {X 0,Y 90.366,Z 446.816,A -85,B 0,C 180,E1 -28796.083,E2 -28796.083} C_VEL
LIN {X 0,Y 91.966,Z 449.9,A -85,B 0,C 180,E1 -28804.519,E2 -28804.519} C_VEL
LIN {X 0,Y 94.356,Z 454.566,A -85,B 0,C 180,E1 -28811.002,E2 -28811.002} C_VEL
LIN {X 0,Y 96.145,Z 457.985,A -85,B 0,C 180,E1 -28814.552,E2 -28814.552} C_VEL
LIN {X 0,Y 99.189,Z 464.116,A -85,B 0,C 180,E1 -28819.467,E2 -28819.467} C_VEL
LIN {X 0,Y 100.984,Z 468.475,A -85,B 0,C 180,E1 -28822.017,E2 -28822.017} C_VEL
LIN {X 0,Y 102.685,Z 476.044,A -85,B 0,C 180,E1 -28824.648,E2 -28824.648} C_VEL
LIN {X 0,Y 102.544,Z 480.106,A -85,B 0,C 180,E1 -28825.056,E2 -28825.056} C_VEL
LIN {X 0,Y 99.509,Z 509.183,A -85,B 0,C 180,E1 -28826.411,E2 -28826.411} C_VEL
LIN {X 0,Y 96.832,Z 522.886,A -85,B 0,C 180,E1 -28827.511,E2 -28827.511} C_VEL
LIN {X 0,Y 93.45,Z 534.918,A -85,B 0,C 180,E1 -28829.044,E2 -28829.044} C_VEL
LIN {X 0,Y 89.906,Z 544.481,A -85,B 0,C 180,E1 -28830.7,E2 -28830.7} C_VEL
LIN {X 0,Y 85.075,Z 555.248,A -85,B 0,C 180,E1 -28833.238,E2 -28833.238} C_VEL
LIN {X 0,Y 81.112,Z 562.829,A -85,B 0,C 180,E1 -28835.68,E2 -28835.68} C_VEL
LIN {X 0,Y 75.594,Z 572.437,A -85,B 0,C 180,E1 -28839.916,E2 -28839.916} C_VEL
LIN {X 0,Y 70.985,Z 579.482,A -85,B 0,C 180,E1 -28844.091,E2 -28844.091} C_VEL
LIN {X 0,Y 65.101,Z 588.375,A -85,B 0,C 180,E1 -28851.631,E2 -28851.631} C_VEL
LIN {X 0,Y 60.454,Z 595.405,A -85,B 0,C 180,E1 -28860.392,E2 -28860.392} C_VEL
LIN {X 0,Y 56.991,Z 601.831,A -85,B 0,C 180,E1 -28872.044,E2 -28872.044} C_VEL
LIN {X 0,Y 55.873,Z 606.012,A -85,B 0,C 180,E1 -28882.774,E2 -28882.774} C_VEL
LIN {X 0,Y 55.902,Z 608.184,A -85,B 0,C 180,E1 -28890,E2 -28890} C_VEL
LIN {X 0,Y 55.887,Z 609.807,A -85,B 0,C 180,E1 -28897.224,E2 -28897.224} C_VEL
LIN {X 0,Y 57.832,Z 611.838,A -85,B 0,C 180,E1 -28911.381,E2 -28911.381} C_VEL
LIN {X 0,Y 59.973,Z 612.281,A -85,B 0,C 180,E1 -28917.952,E2 -28917.952} C_VEL
LIN {X 0,Y 66.511,Z 611.973,A -85,B 0,C 180,E1 -28929.345,E2 -28929.345} C_VEL
LIN {X 0,Y 75.245,Z 610.172,A -85,B 0,C 180,E1 -28938.348,E2 -28938.348} C_VEL
LIN {X 0,Y 80.692,Z 608.489,A -85,B 0,C 180,E1 -28942.435,E2 -28942.435} C_VEL
LIN {X 0,Y 90.93,Z 604.403,A -85,B 0,C 180,E1 -28948.231,E2 -28948.231} C_VEL
LIN {X 0,Y 99.628,Z 600.018,A -85,B 0,C 180,E1 -28951.856,E2 -28951.856} C_VEL
LIN {X 0,Y 110.252,Z 593.457,A -85,B 0,C 180,E1 -28955.277,E2 -28955.277} C_VEL
LIN {X 0,Y 119.692,Z 586.294,A -85,B 0,C 180,E1 -28957.635,E2 -28957.635} C_VEL
LIN {X 0,Y 129.281,Z 577.439,A -85,B 0,C 180,E1 -28959.673,E2 -28959.673} C_VEL
LIN {X 0,Y 137.428,Z 568.379,A -85,B 0,C 180,E1 -28961.095,E2 -28961.095} C_VEL
LIN {X 0,Y 144.869,Z 558.389,A -85,B 0,C 180,E1 -28962.183,E2 -28962.183} C_VEL
LIN {X 0,Y 151.513,Z 547.335,A -85,B 0,C 180,E1 -28963.074,E2 -28963.074} C_VEL
LIN {X 0,Y 157.447,Z 534.789,A -85,B 0,C 180,E1 -28963.784,E2 -28963.784} C_VEL
LIN {X 0,Y 160.708,Z 525.856,A -85,B 0,C 180,E1 -28964.169,E2 -28964.169} C_VEL
LIN {X 0,Y 161.209,Z 523.936,A -85,B 0,C 180,E1 -28964.529,E2 -28964.529} C_VEL
LIN {X 0,Y 161.168,Z 520.777,A -85,B 0,C 180,E1 -28967.407,E2 -28967.407} C_VEL
LIN {X 0,Y 161.12,Z 518.385,A -85,B 0,C 180,E1 -28971.851,E2 -28971.851} C_VEL
LIN {X 0,Y 161.093,Z 518.58,A -85,B 0,C 180,E1 -28974.158,E2 -28974.158} C_VEL
LIN {X 0,Y 161.228,Z 522.365,A -85,B 0,C 180,E1 -28980.001,E2 -28980.001} C_VEL
LIN {X 0,Y 161.278,Z 522.804,A -85,B 0,C 180,E1 -28980.535,E2 -28980.535} C_VEL
LIN {X 0,Y 156.886,Z 534.666,A -85,B 0,C 180,E1 -28981.195,E2 -28981.195} C_VEL
LIN {X 0,Y 151.203,Z 546.413,A -85,B 0,C 180,E1 -28982.128,E2 -28982.128} C_VEL
LIN {X 0,Y 144.794,Z 556.83,A -85,B 0,C 180,E1 -28983.21,E2 -28983.21} C_VEL
LIN {X 0,Y 141.253,Z 561.601,A -85,B 0,C 180,E1 -28983.529,E2 -28983.529} C_VEL
LIN {X 0,Y 134.68,Z 569.099,A -85,B 0,C 180,E1 -28983.432,E2 -28983.432} C_VEL
LIN {X 0,Y 127.656,Z 575.979,A -85,B 0,C 180,E1 -28983.438,E2 -28983.438} C_VEL
LIN {X 0,Y 123.42,Z 579.799,A -85,B 0,C 180,E1 -28983.979,E2 -28983.979} C_VEL
LIN {X 0,Y 114.808,Z 586.769,A -85,B 0,C 180,E1 -28985.887,E2 -28985.887} C_VEL
LIN {X 0,Y 106.475,Z 592.408,A -85,B 0,C 180,E1 -28988.083,E2 -28988.083} C_VEL
LIN {X 0,Y 96.724,Z 597.853,A -85,B 0,C 180,E1 -28991.219,E2 -28991.219} C_VEL
LIN {X 0,Y 87.306,Z 602.024,A -85,B 0,C 180,E1 -28994.993,E2 -28994.993} C_VEL
LIN {X 0,Y 81.281,Z 604.148,A -85,B 0,C 180,E1 -28997.993,E2 -28997.993} C_VEL
LIN {X 0,Y 74.38,Z 606.089,A -85,B 0,C 180,E1 -29002.209,E2 -29002.209} C_VEL
LIN {X 0,Y 64.967,Z 607.769,A -85,B 0,C 180,E1 -29010.071,E2 -29010.071} C_VEL
LIN {X 0,Y 60.216,Z 608.084,A -85,B 0,C 180,E1 -29015.704,E2 -29015.704} C_VEL
LIN {X 0,Y 56.361,Z 607.986,A -85,B 0,C 180,E1 -29021.569,E2 -29021.569} C_VEL
LIN {X 0,Y 53.036,Z 607.47,A -85,B 0,C 180,E1 -29028.506,E2 -29028.506} C_VEL
LIN {X 0,Y 50.343,Z 606.382,A -85,B 0,C 180,E1 -29036.894,E2 -29036.894} C_VEL
LIN {X 0,Y 48.894,Z 605.099,A -85,B 0,C 180,E1 -29044.456,E2 -29044.456} C_VEL
LIN {X 0,Y 48.273,Z 602.176,A -85,B 0,C 180,E1 -29057.386,E2 -29057.386} C_VEL
LIN {X 0,Y 49.757,Z 598.196,A -85,B 0,C 180,E1 -29070,E2 -29070} C_VEL
LIN {X 0,Y 53.023,Z 593.075,A -85,B 0,C 180,E1 -29081.468,E2 -29081.468} C_VEL
LIN {X 0,Y 57.788,Z 586.665,A -85,B 0,C 180,E1 -29091.398,E2 -29091.398} C_VEL
LIN {X 0,Y 63.845,Z 578.632,A -85,B 0,C 180,E1 -29099.692,E2 -29099.692} C_VEL
LIN {X 0,Y 69.736,Z 570.242,A -85,B 0,C 180,E1 -29105.628,E2 -29105.628} C_VEL
LIN {X 0,Y 75.863,Z 560.497,A -85,B 0,C 180,E1 -29110.426,E2 -29110.426} C_VEL
LIN {X 0,Y 81.999,Z 549.233,A -85,B 0,C 180,E1 -29114.136,E2 -29114.136} C_VEL
LIN {X 0,Y 86.868,Z 538.228,A -85,B 0,C 180,E1 -29116.729,E2 -29116.729} C_VEL
LIN {X 0,Y 91.173,Z 526.05,A -85,B 0,C 180,E1 -29118.725,E2 -29118.725} C_VEL
LIN {X 0,Y 94.514,Z 512.893,A -85,B 0,C 180,E1 -29120.195,E2 -29120.195} C_VEL
LIN {X 0,Y 96.716,Z 498.979,A -85,B 0,C 180,E1 -29121.147,E2 -29121.147} C_VEL
LIN {X 0,Y 99.069,Z 476.014,A -85,B 0,C 180,E1 -29122.172,E2 -29122.172} C_VEL
LIN {X 0,Y 96.54,Z 469.508,A -85,B 0,C 180,E1 -29126.117,E2 -29126.117} C_VEL
LIN {X 0,Y 93.74,Z 463.386,A -85,B 0,C 180,E1 -29131.355,E2 -29131.355} C_VEL
LIN {X 0,Y 91.775,Z 459.547,A -85,B 0,C 180,E1 -29136.146,E2 -29136.146} C_VEL
LIN {X 0,Y 90.465,Z 456.701,A -85,B 0,C 180,E1 -29140.72,E2 -29140.72} C_VEL
LIN {X 0,Y 89.233,Z 453.871,A -85,B 0,C 180,E1 -29150.936,E2 -29150.936} C_VEL
LIN {X 0,Y 89.434,Z 453.929,A -85,B 0,C 180,E1 -29155.767,E2 -29155.767} C_VEL
LIN {X 0,Y 90.72,Z 456.785,A -85,B 0,C 180,E1 -29163.469,E2 -29163.469} C_VEL
LIN {X 0,Y 92.584,Z 460.855,A -85,B 0,C 180,E1 -29169.257,E2 -29169.257} C_VEL
LIN {X 0,Y 94.413,Z 464.748,A -85,B 0,C 180,E1 -29173.339,E2 -29173.339} C_VEL
LIN {X 0,Y 97.016,Z 470.612,A -85,B 0,C 180,E1 -29177.987,E2 -29177.987} C_VEL
LIN {X 0,Y 97.975,Z 473.495,A -85,B 0,C 180,E1 -29179.589,E2 -29179.589} C_VEL
LIN {X 0,Y 98.979,Z 478.62,A -85,B 0,C 180,E1 -29181.465,E2 -29181.465} C_VEL
LIN {X 0,Y 95.733,Z 509.001,A -85,B 0,C 180,E1 -29182.892,E2 -29182.892} C_VEL
LIN {X 0,Y 93.102,Z 521.951,A -85,B 0,C 180,E1 -29183.851,E2 -29183.851} C_VEL
LIN {X 0,Y 89.447,Z 534.526,A -85,B 0,C 180,E1 -29185.371,E2 -29185.371} C_VEL
LIN {X 0,Y 85.739,Z 544.102,A -85,B 0,C 180,E1 -29186.951,E2 -29186.951} C_VEL
LIN {X 0,Y 80.671,Z 554.884,A -85,B 0,C 180,E1 -29189.405,E2 -29189.405} C_VEL
LIN {X 0,Y 76.453,Z 562.46,A -85,B 0,C 180,E1 -29191.756,E2 -29191.756} C_VEL
LIN {X 0,Y 69.951,Z 573.058,A -85,B 0,C 180,E1 -29196.51,E2 -29196.51} C_VEL
LIN {X 0,Y 64.969,Z 579.977,A -85,B 0,C 180,E1 -29200.782,E2 -29200.782} C_VEL
LIN {X 0,Y 59.635,Z 587.345,A -85,B 0,C 180,E1 -29207.342,E2 -29207.342} C_VEL
LIN {X 0,Y 54.369,Z 594.55,A -85,B 0,C 180,E1 -29216.677,E2 -29216.677} C_VEL
LIN {X 0,Y 50.259,Z 601.081,A -85,B 0,C 180,E1 -29229.538,E2 -29229.538} C_VEL
LIN {X 0,Y 48.827,Z 605.359,A -85,B 0,C 180,E1 -29241.724,E2 -29241.724} C_VEL
LIN {X 0,Y 48.817,Z 607.594,A -85,B 0,C 180,E1 -29250,E2 -29250} C_VEL
LIN {X 0,Y 48.864,Z 609.288,A -85,B 0,C 180,E1 -29258.269,E2 -29258.269} C_VEL
LIN {X 0,Y 51.269,Z 611.4,A -85,B 0,C 180,E1 -29274.282,E2 -29274.282} C_VEL
LIN {X 0,Y 57.113,Z 611.997,A -85,B 0,C 180,E1 -29287.97,E2 -29287.97} C_VEL
LIN {X 0,Y 65.705,Z 611.031,A -85,B 0,C 180,E1 -29298.48,E2 -29298.48} C_VEL
LIN {X 0,Y 75.998,Z 608.565,A -85,B 0,C 180,E1 -29306.332,E2 -29306.332} C_VEL
LIN {X 0,Y 84.458,Z 605.617,A -85,B 0,C 180,E1 -29310.893,E2 -29310.893} C_VEL
LIN {X 0,Y 93.414,Z 601.681,A -85,B 0,C 180,E1 -29314.528,E2 -29314.528} C_VEL
LIN {X 0,Y 102.718,Z 596.654,A -85,B 0,C 180,E1 -29317.466,E2 -29317.466} C_VEL
LIN {X 0,Y 112.273,Z 590.383,A -85,B 0,C 180,E1 -29319.875,E2 -29319.875} C_VEL
LIN {X 0,Y 122.076,Z 582.574,A -85,B 0,C 180,E1 -29321.785,E2 -29321.785} C_VEL
LIN {X 0,Y 131.963,Z 572.879,A -85,B 0,C 180,E1 -29323.457,E2 -29323.457} C_VEL
LIN {X 0,Y 140.34,Z 562.862,A -85,B 0,C 180,E1 -29324.576,E2 -29324.576} C_VEL
LIN {X 0,Y 147.925,Z 551.557,A -85,B 0,C 180,E1 -29325.467,E2 -29325.467} C_VEL
LIN {X 0,Y 154.297,Z 539.588,A -85,B 0,C 180,E1 -29326.145,E2 -29326.145} C_VEL
LIN {X 0,Y 158.261,Z 530.094,A -85,B 0,C 180,E1 -29326.528,E2 -29326.528} C_VEL
LIN {X 0,Y 158.804,Z 528.476,A -85,B 0,C 180,E1 -29326.807,E2 -29326.807} C_VEL
LIN {X 0,Y 158.844,Z 526.326,A -85,B 0,C 180,E1 -29329.807,E2 -29329.807} C_VEL
LIN {X 0,Y 159.007,Z 525.083,A -85,B 0,C 180,E1 -29332.381,E2 -29332.381} C_VEL
LIN {X 0,Y 158.809,Z 525.989,A -85,B 0,C 180,E1 -29334.923,E2 -29334.923} C_VEL
LIN {X 0,Y 158.686,Z 527.897,A -85,B 0,C 180,E1 -29338.097,E2 -29338.097} C_VEL
LIN {X 0,Y 158.226,Z 529.229,A -85,B 0,C 180,E1 -29338.33,E2 -29338.33} C_VEL
LIN {X 0,Y 152.877,Z 541.479,A -85,B 0,C 180,E1 -29339.044,E2 -29339.044} C_VEL
LIN {X 0,Y 146.568,Z 552.64,A -85,B 0,C 180,E1 -29340.001,E2 -29340.001} C_VEL
LIN {X 0,Y 138.829,Z 563.511,A -85,B 0,C 180,E1 -29341.171,E2 -29341.171} C_VEL
LIN {X 0,Y 130.152,Z 573.414,A -85,B 0,C 180,E1 -29342.665,E2 -29342.665} C_VEL
LIN {X 0,Y 123.42,Z 579.799,A -85,B 0,C 180,E1 -29343.979,E2 -29343.979} C_VEL
LIN {X 0,Y 118.988,Z 583.491,A -85,B 0,C 180,E1 -29344.597,E2 -29344.597} C_VEL
LIN {X 0,Y 110.871,Z 589.179,A -85,B 0,C 180,E1 -29344.892,E2 -29344.892} C_VEL
LIN {X 0,Y 102.36,Z 594.186,A -85,B 0,C 180,E1 -29345.32,E2 -29345.32} C_VEL
LIN {X 0,Y 97.346,Z 596.808,A -85,B 0,C 180,E1 -29346.275,E2 -29346.275} C_VEL
LIN {X 0,Y 85.678,Z 601.997,A -85,B 0,C 180,E1 -29350.161,E2 -29350.161} C_VEL
LIN {X 0,Y 79.292,Z 604.225,A -85,B 0,C 180,E1 -29352.85,E2 -29352.85} C_VEL
LIN {X 0,Y 70.773,Z 606.488,A -85,B 0,C 180,E1 -29357.334,E2 -29357.334} C_VEL
LIN {X 0,Y 61.553,Z 608.04,A -85,B 0,C 180,E1 -29364.021,E2 -29364.021} C_VEL
LIN {X 0,Y 55.245,Z 608.431,A -85,B 0,C 180,E1 -29370.59,E2 -29370.59} C_VEL
LIN {X 0,Y 47.704,Z 607.909,A -85,B 0,C 180,E1 -29382.556,E2 -29382.556} C_VEL
LIN {X 0,Y 43.896,Z 606.692,A -85,B 0,C 180,E1 -29393.186,E2 -29393.186} C_VEL
LIN {X 0,Y 41.206,Z 603.91,A -85,B 0,C 180,E1 -29410.056,E2 -29410.056} C_VEL
LIN {X 0,Y 41.754,Z 600.429,A -85,B 0,C 180,E1 -29425.027,E2 -29425.027} C_VEL
LIN {X 0,Y 44.588,Z 595.779,A -85,B 0,C 180,E1 -29439.069,E2 -29439.069} C_VEL
LIN {X 0,Y 49.249,Z 589.95,A -85,B 0,C 180,E1 -29450.901,E2 -29450.901} C_VEL
LIN {X 0,Y 55.436,Z 582.637,A -85,B 0,C 180,E1 -29460.471,E2 -29460.471} C_VEL
LIN {X 0,Y 62.201,Z 574.133,A -85,B 0,C 180,E1 -29467.725,E2 -29467.725} C_VEL
LIN {X 0,Y 69.26,Z 564.244,A -85,B 0,C 180,E1 -29473.23,E2 -29473.23} C_VEL
LIN {X 0,Y 75.568,Z 553.838,A -85,B 0,C 180,E1 -29477.086,E2 -29477.086} C_VEL
LIN {X 0,Y 81.391,Z 542.294,A -85,B 0,C 180,E1 -29480.025,E2 -29480.025} C_VEL
LIN {X 0,Y 86.237,Z 530.204,A -85,B 0,C 180,E1 -29482.137,E2 -29482.137} C_VEL
LIN {X 0,Y 90.125,Z 517.104,A -85,B 0,C 180,E1 -29483.652,E2 -29483.652} C_VEL
LIN {X 0,Y 92.68,Z 504.202,A -85,B 0,C 180,E1 -29484.655,E2 -29484.655} C_VEL
LIN {X 0,Y 95.517,Z 478.955,A -85,B 0,C 180,E1 -29485.75,E2 -29485.75} C_VEL
LIN {X 0,Y 93.431,Z 473.412,A -85,B 0,C 180,E1 -29489.684,E2 -29489.684} C_VEL
LIN {X 0,Y 91.507,Z 468.865,A -85,B 0,C 180,E1 -29494.106,E2 -29494.106} C_VEL
LIN {X 0,Y 90.194,Z 465.822,A -85,B 0,C 180,E1 -29498.035,E2 -29498.035} C_VEL
LIN {X 0,Y 89.194,Z 463.427,A -85,B 0,C 180,E1 -29502.216,E2 -29502.216} C_VEL
LIN {X 0,Y 88.332,Z 461.073,A -85,B 0,C 180,E1 -29510.843,E2 -29510.843} C_VEL
LIN {X 0,Y 88.534,Z 461.286,A -85,B 0,C 180,E1 -29516.002,E2 -29516.002} C_VEL
LIN {X 0,Y 89.421,Z 463.406,A -85,B 0,C 180,E1 -29521.969,E2 -29521.969} C_VEL
LIN {X 0,Y 91.116,Z 467.659,A -85,B 0,C 180,E1 -29528.071,E2 -29528.071} C_VEL
LIN {X 0,Y 92.815,Z 471.7,A -85,B 0,C 180,E1 -29532.282,E2 -29532.282} C_VEL
LIN {X 0,Y 94.893,Z 477.198,A -85,B 0,C 180,E1 -29536.452,E2 -29536.452} C_VEL
LIN {X 0,Y 95.504,Z 480.437,A -85,B 0,C 180,E1 -29537.811,E2 -29537.811} C_VEL
LIN {X 0,Y 92.351,Z 508.765,A -85,B 0,C 180,E1 -29539.105,E2 -29539.105} C_VEL
LIN {X 0,Y 89.726,Z 521.306,A -85,B 0,C 180,E1 -29539.964,E2 -29539.964} C_VEL
LIN {X 0,Y 85.845,Z 534.111,A -85,B 0,C 180,E1 -29541.372,E2 -29541.372} C_VEL
LIN {X 0,Y 81.974,Z 543.706,A -85,B 0,C 180,E1 -29542.835,E2 -29542.835} C_VEL
LIN {X 0,Y 76.667,Z 554.506,A -85,B 0,C 180,E1 -29545.148,E2 -29545.148} C_VEL
LIN {X 0,Y 72.209,Z 562.085,A -85,B 0,C 180,E1 -29547.364,E2 -29547.364} C_VEL
LIN {X 0,Y 65.925,Z 571.716,A -85,B 0,C 180,E1 -29551.479,E2 -29551.479} C_VEL
LIN {X 0,Y 60.573,Z 578.805,A -85,B 0,C 180,E1 -29555.693,E2 -29555.693} C_VEL
LIN {X 0,Y 53.489,Z 587.676,A -85,B 0,C 180,E1 -29563.727,E2 -29563.727} C_VEL
LIN {X 0,Y 47.665,Z 594.713,A -85,B 0,C 180,E1 -29573.859,E2 -29573.859} C_VEL
LIN {X 0,Y 43.617,Z 600.326,A -85,B 0,C 180,E1 -29586.245,E2 -29586.245} C_VEL
LIN {X 0,Y 41.797,Z 604.705,A -85,B 0,C 180,E1 -29600.32,E2 -29600.32} C_VEL
LIN {X 0,Y 41.733,Z 606.988,A -85,B 0,C 180,E1 -29610,E2 -29610} C_VEL
LIN {X 0,Y 41.841,Z 608.755,A -85,B 0,C 180,E1 -29619.669,E2 -29619.669} C_VEL
LIN {X 0,Y 44.881,Z 610.958,A -85,B 0,C 180,E1 -29638.019,E2 -29638.019} C_VEL
LIN {X 0,Y 51.695,Z 611.653,A -85,B 0,C 180,E1 -29652.824,E2 -29652.824} C_VEL
LIN {X 0,Y 56.228,Z 611.432,A -85,B 0,C 180,E1 -29658.585,E2 -29658.585} C_VEL
LIN {X 0,Y 66.624,Z 609.808,A -85,B 0,C 180,E1 -29667.551,E2 -29667.551} C_VEL
LIN {X 0,Y 78.204,Z 606.653,A -85,B 0,C 180,E1 -29673.982,E2 -29673.982} C_VEL
LIN {X 0,Y 87.435,Z 603.152,A -85,B 0,C 180,E1 -29677.57,E2 -29677.57} C_VEL
LIN {X 0,Y 96.98,Z 598.605,A -85,B 0,C 180,E1 -29680.402,E2 -29680.402} C_VEL
LIN {X 0,Y 108.407,Z 591.773,A -85,B 0,C 180,E1 -29682.982,E2 -29682.982} C_VEL
LIN {X 0,Y 118.376,Z 584.396,A -85,B 0,C 180,E1 -29684.74,E2 -29684.74} C_VEL
LIN {X 0,Y 128.458,Z 575.276,A -85,B 0,C 180,E1 -29686.189,E2 -29686.189} C_VEL
LIN {X 0,Y 136.931,Z 565.833,A -85,B 0,C 180,E1 -29687.202,E2 -29687.202} C_VEL
LIN {X 0,Y 144.61,Z 555.386,A -85,B 0,C 180,E1 -29687.972,E2 -29687.972} C_VEL
LIN {X 0,Y 151.221,Z 544.236,A -85,B 0,C 180,E1 -29688.574,E2 -29688.574} C_VEL
LIN {X 0,Y 155.849,Z 534.432,A -85,B 0,C 180,E1 -29688.953,E2 -29688.953} C_VEL
LIN {X 0,Y 156.243,Z 533.229,A -85,B 0,C 180,E1 -29689.635,E2 -29689.635} C_VEL
LIN {X 0,Y 156.484,Z 531.885,A -85,B 0,C 180,E1 -29692.257,E2 -29692.257} C_VEL
LIN {X 0,Y 156.099,Z 533.24,A -85,B 0,C 180,E1 -29695.837,E2 -29695.837} C_VEL
LIN {X 0,Y 153.387,Z 539.268,A -85,B 0,C 180,E1 -29696.242,E2 -29696.242} C_VEL
LIN {X 0,Y 146.76,Z 551.337,A -85,B 0,C 180,E1 -29697.093,E2 -29697.093} C_VEL
LIN {X 0,Y 139.763,Z 561.455,A -85,B 0,C 180,E1 -29698.002,E2 -29698.002} C_VEL
LIN {X 0,Y 131.788,Z 570.837,A -85,B 0,C 180,E1 -29699.112,E2 -29699.112} C_VEL
LIN {X 0,Y 122.886,Z 579.457,A -85,B 0,C 180,E1 -29700.554,E2 -29700.554} C_VEL
LIN {X 0,Y 112.554,Z 587.641,A -85,B 0,C 180,E1 -29702.522,E2 -29702.522} C_VEL
LIN {X 0,Y 102.282,Z 594.171,A -85,B 0,C 180,E1 -29704.928,E2 -29704.928} C_VEL
LIN {X 0,Y 97.346,Z 596.808,A -85,B 0,C 180,E1 -29706.275,E2 -29706.275} C_VEL
LIN {X 0,Y 92.24,Z 599.227,A -85,B 0,C 180,E1 -29707.377,E2 -29707.377} C_VEL
LIN {X 0,Y 83.078,Z 602.747,A -85,B 0,C 180,E1 -29708.396,E2 -29708.396} C_VEL
LIN {X 0,Y 73.75,Z 605.483,A -85,B 0,C 180,E1 -29709.742,E2 -29709.742} C_VEL
LIN {X 0,Y 68.475,Z 606.716,A -85,B 0,C 180,E1 -29711.595,E2 -29711.595} C_VEL
LIN {X 0,Y 58.9,Z 608.276,A -85,B 0,C 180,E1 -29717.342,E2 -29717.342} C_VEL
LIN {X 0,Y 50.782,Z 608.778,A -85,B 0,C 180,E1 -29724.533,E2 -29724.533} C_VEL
LIN {X 0,Y 43.005,Z 608.333,A -85,B 0,C 180,E1 -29735.206,E2 -29735.206} C_VEL
LIN {X 0,Y 37.625,Z 606.985,A -85,B 0,C 180,E1 -29748.35,E2 -29748.35} C_VEL
LIN {X 0,Y 34.043,Z 603.509,A -85,B 0,C 180,E1 -29771.961,E2 -29771.961} C_VEL
LIN {X 0,Y 35.182,Z 599.732,A -85,B 0,C 180,E1 -29790,E2 -29790} C_VEL
LIN {X 0,Y 38.969,Z 594.829,A -85,B 0,C 180,E1 -29805.695,E2 -29805.695} C_VEL
LIN {X 0,Y 44.708,Z 588.668,A -85,B 0,C 180,E1 -29818.137,E2 -29818.137} C_VEL
LIN {X 0,Y 51.88,Z 581.016,A -85,B 0,C 180,E1 -29827.559,E2 -29827.559} C_VEL
LIN {X 0,Y 58.941,Z 572.695,A -85,B 0,C 180,E1 -29833.989,E2 -29833.989} C_VEL
LIN {X 0,Y 65.678,Z 563.674,A -85,B 0,C 180,E1 -29838.506,E2 -29838.506} C_VEL
LIN {X 0,Y 72.413,Z 553.07,A -85,B 0,C 180,E1 -29842.05,E2 -29842.05} C_VEL
LIN {X 0,Y 78.573,Z 541.25,A -85,B 0,C 180,E1 -29844.704,E2 -29844.704} C_VEL
LIN {X 0,Y 83.632,Z 528.619,A -85,B 0,C 180,E1 -29846.623,E2 -29846.623} C_VEL
LIN {X 0,Y 87.492,Z 515.505,A -85,B 0,C 180,E1 -29847.969,E2 -29847.969} C_VEL
LIN {X 0,Y 89.87,Z 503.221,A -85,B 0,C 180,E1 -29848.757,E2 -29848.757} C_VEL
LIN {X 0,Y 92.264,Z 482.735,A -85,B 0,C 180,E1 -29849.534,E2 -29849.534} C_VEL
LIN {X 0,Y 92.119,Z 481.605,A -85,B 0,C 180,E1 -29850.001,E2 -29850.001} C_VEL
LIN {X 0,Y 90.532,Z 476.942,A -85,B 0,C 180,E1 -29853.924,E2 -29853.924} C_VEL
LIN {X 0,Y 88.855,Z 472.475,A -85,B 0,C 180,E1 -29859.401,E2 -29859.401} C_VEL
LIN {X 0,Y 87.99,Z 470.141,A -85,B 0,C 180,E1 -29863.745,E2 -29863.745} C_VEL
LIN {X 0,Y 87.431,Z 468.265,A -85,B 0,C 180,E1 -29870.747,E2 -29870.747} C_VEL
LIN {X 0,Y 87.603,Z 468.394,A -85,B 0,C 180,E1 -29875.678,E2 -29875.678} C_VEL
LIN {X 0,Y 88.243,Z 470.258,A -85,B 0,C 180,E1 -29880.801,E2 -29880.801} C_VEL
LIN {X 0,Y 89.623,Z 474.221,A -85,B 0,C 180,E1 -29886.613,E2 -29886.613} C_VEL
LIN {X 0,Y 91.474,Z 479.477,A -85,B 0,C 180,E1 -29891.776,E2 -29891.776} C_VEL
LIN {X 0,Y 92.403,Z 482.721,A -85,B 0,C 180,E1 -29893.993,E2 -29893.993} C_VEL
LIN {X 0,Y 89.29,Z 508.847,A -85,B 0,C 180,E1 -29895.06,E2 -29895.06} C_VEL
LIN {X 0,Y 86.318,Z 522.218,A -85,B 0,C 180,E1 -29895.899,E2 -29895.899} C_VEL
LIN {X 0,Y 82.299,Z 534.67,A -85,B 0,C 180,E1 -29897.187,E2 -29897.187} C_VEL
LIN {X 0,Y 77.899,Z 544.975,A -85,B 0,C 180,E1 -29898.687,E2 -29898.687} C_VEL
LIN {X 0,Y 72.325,Z 555.374,A -85,B 0,C 180,E1 -29900.73,E2 -29900.73} C_VEL
LIN {X 0,Y 67.701,Z 562.846,A -85,B 0,C 180,E1 -29902.885,E2 -29902.885} C_VEL
LIN {X 0,Y 60.398,Z 573.105,A -85,B 0,C 180,E1 -29907.286,E2 -29907.286} C_VEL
LIN {X 0,Y 52.458,Z 582.452,A -85,B 0,C 180,E1 -29913.455,E2 -29913.455} C_VEL
LIN {X 0,Y 45.325,Z 590.432,A -85,B 0,C 180,E1 -29922.565,E2 -29922.565} C_VEL
LIN {X 0,Y 40.214,Z 595.868,A -85,B 0,C 180,E1 -29932.29,E2 -29932.29} C_VEL
LIN {X 0,Y 36.086,Z 601.183,A -85,B 0,C 180,E1 -29947.076,E2 -29947.076} C_VEL
LIN {X 0,Y 34.569,Z 605.274,A -85,B 0,C 180,E1 -29964.166,E2 -29964.166} C_VEL
LIN {X 0,Y 34.65,Z 606.365,A -85,B 0,C 180,E1 -29970,E2 -29970} C_VEL
LIN {X 0,Y 34.872,Z 608.183,A -85,B 0,C 180,E1 -29981.627,E2 -29981.627} C_VEL
LIN {X 0,Y 36.187,Z 609.562,A -85,B 0,C 180,E1 -29992.856,E2 -29992.856} C_VEL
LIN {X 0,Y 42.274,Z 611.085,A -85,B 0,C 180,E1 -30011.681,E2 -30011.681} C_VEL
LIN {X 0,Y 51.784,Z 611.138,A -85,B 0,C 180,E1 -30024.517,E2 -30024.517} C_VEL
LIN {X 0,Y 63.085,Z 609.626,A -85,B 0,C 180,E1 -30033.027,E2 -30033.027} C_VEL
LIN {X 0,Y 75.353,Z 606.57,A -85,B 0,C 180,E1 -30038.852,E2 -30038.852} C_VEL
LIN {X 0,Y 84.974,Z 603.158,A -85,B 0,C 180,E1 -30042.01,E2 -30042.01} C_VEL
LIN {X 0,Y 94.832,Z 598.711,A -85,B 0,C 180,E1 -30044.451,E2 -30044.451} C_VEL
LIN {X 0,Y 106.543,Z 592.048,A -85,B 0,C 180,E1 -30046.641,E2 -30046.641} C_VEL
LIN {X 0,Y 116.71,Z 584.8,A -85,B 0,C 180,E1 -30048.101,E2 -30048.101} C_VEL
LIN {X 0,Y 125.239,Z 577.467,A -85,B 0,C 180,E1 -30049.118,E2 -30049.118} C_VEL
LIN {X 0,Y 133.82,Z 568.609,A -85,B 0,C 180,E1 -30049.963,E2 -30049.963} C_VEL
LIN {X 0,Y 142.449,Z 557.72,A -85,B 0,C 180,E1 -30050.65,E2 -30050.65} C_VEL
LIN {X 0,Y 149.355,Z 546.76,A -85,B 0,C 180,E1 -30051.17,E2 -30051.17} C_VEL
LIN {X 0,Y 152.967,Z 539.862,A -85,B 0,C 180,E1 -30051.405,E2 -30051.405} C_VEL
LIN {X 0,Y 153.56,Z 538.547,A -85,B 0,C 180,E1 -30052.109,E2 -30052.109} C_VEL
LIN {X 0,Y 153.439,Z 538.708,A -85,B 0,C 180,E1 -30053.197,E2 -30053.197} C_VEL
LIN {X 0,Y 153.213,Z 539.171,A -85,B 0,C 180,E1 -30053.575,E2 -30053.575} C_VEL
LIN {X 0,Y 147.288,Z 550.018,A -85,B 0,C 180,E1 -30054.202,E2 -30054.202} C_VEL
LIN {X 0,Y 140.221,Z 560.395,A -85,B 0,C 180,E1 -30054.957,E2 -30054.957} C_VEL
LIN {X 0,Y 132.109,Z 570.094,A -85,B 0,C 180,E1 -30055.907,E2 -30055.907} C_VEL
LIN {X 0,Y 122.482,Z 579.385,A -85,B 0,C 180,E1 -30057.18,E2 -30057.18} C_VEL
LIN {X 0,Y 112.473,Z 587.243,A -85,B 0,C 180,E1 -30058.733,E2 -30058.733} C_VEL
LIN {X 0,Y 101.912,Z 593.955,A -85,B 0,C 180,E1 -30060.75,E2 -30060.75} C_VEL
LIN {X 0,Y 91.505,Z 599.195,A -85,B 0,C 180,E1 -30063.203,E2 -30063.203} C_VEL
LIN {X 0,Y 81.307,Z 603.186,A -85,B 0,C 180,E1 -30066.275,E2 -30066.275} C_VEL
LIN {X 0,Y 68.475,Z 606.716,A -85,B 0,C 180,E1 -30071.595,E2 -30071.595} C_VEL
LIN {X 0,Y 63.222,Z 607.716,A -85,B 0,C 180,E1 -30073.783,E2 -30073.783} C_VEL
LIN {X 0,Y 53.821,Z 608.754,A -85,B 0,C 180,E1 -30076.704,E2 -30076.704} C_VEL
LIN {X 0,Y 44.541,Z 609.074,A -85,B 0,C 180,E1 -30080.83,E2 -30080.83} C_VEL
LIN {X 0,Y 39.709,Z 608.793,A -85,B 0,C 180,E1 -30085.48,E2 -30085.48} C_VEL
LIN {X 0,Y 31.723,Z 607.277,A -85,B 0,C 180,E1 -30101.658,E2 -30101.658} C_VEL
LIN {X 0,Y 27.129,Z 604.174,A -85,B 0,C 180,E1 -30127.134,E2 -30127.134} C_VEL
LIN {X 0,Y 28.131,Z 600.081,A -85,B 0,C 180,E1 -30152.019,E2 -30152.019} C_VEL
LIN {X 0,Y 32.058,Z 595.703,A -85,B 0,C 180,E1 -30169.198,E2 -30169.198} C_VEL
LIN {X 0,Y 38.533,Z 589.657,A -85,B 0,C 180,E1 -30183.172,E2 -30183.172} C_VEL
LIN {X 0,Y 46.41,Z 582.142,A -85,B 0,C 180,E1 -30192.955,E2 -30192.955} C_VEL
LIN {X 0,Y 54.105,Z 573.93,A -85,B 0,C 180,E1 -30199.296,E2 -30199.296} C_VEL
LIN {X 0,Y 61.198,Z 565.229,A -85,B 0,C 180,E1 -30203.5,E2 -30203.5} C_VEL
LIN {X 0,Y 68.26,Z 554.906,A -85,B 0,C 180,E1 -30206.775,E2 -30206.775} C_VEL
LIN {X 0,Y 74.649,Z 543.459,A -85,B 0,C 180,E1 -30209.212,E2 -30209.212} C_VEL
LIN {X 0,Y 79.928,Z 531.549,A -85,B 0,C 180,E1 -30210.9,E2 -30210.9} C_VEL
LIN {X 0,Y 84.218,Z 518.363,A -85,B 0,C 180,E1 -30212.132,E2 -30212.132} C_VEL
LIN {X 0,Y 87.051,Z 505.389,A -85,B 0,C 180,E1 -30212.945,E2 -30212.945} C_VEL
LIN {X 0,Y 89.524,Z 485.478,A -85,B 0,C 180,E1 -30213.685,E2 -30213.685} C_VEL
LIN {X 0,Y 88.12,Z 480.964,A -85,B 0,C 180,E1 -30218.353,E2 -30218.353} C_VEL
LIN {X 0,Y 87.391,Z 478.607,A -85,B 0,C 180,E1 -30221.698,E2 -30221.698} C_VEL
LIN {X 0,Y 86.947,Z 477.037,A -85,B 0,C 180,E1 -30224.61,E2 -30224.61} C_VEL
LIN {X 0,Y 86.529,Z 475.481,A -85,B 0,C 180,E1 -30230.65,E2 -30230.65} C_VEL
LIN {X 0,Y 86.69,Z 475.598,A -85,B 0,C 180,E1 -30235.633,E2 -30235.633} C_VEL
LIN {X 0,Y 87.101,Z 477.052,A -85,B 0,C 180,E1 -30239.554,E2 -30239.554} C_VEL
LIN {X 0,Y 88.086,Z 480.52,A -85,B 0,C 180,E1 -30244.718,E2 -30244.718} C_VEL
LIN {X 0,Y 89.577,Z 485.574,A -85,B 0,C 180,E1 -30249.767,E2 -30249.767} C_VEL
LIN {X 0,Y 89.159,Z 489.958,A -85,B 0,C 180,E1 -30250.088,E2 -30250.088} C_VEL
LIN {X 0,Y 86.679,Z 509.054,A -85,B 0,C 180,E1 -30250.753,E2 -30250.753} C_VEL
LIN {X 0,Y 83.572,Z 522.463,A -85,B 0,C 180,E1 -30251.5,E2 -30251.5} C_VEL
LIN {X 0,Y 79.222,Z 535.151,A -85,B 0,C 180,E1 -30252.625,E2 -30252.625} C_VEL
LIN {X 0,Y 74.268,Z 546.106,A -85,B 0,C 180,E1 -30254.085,E2 -30254.085} C_VEL
LIN {X 0,Y 68.467,Z 556.214,A -85,B 0,C 180,E1 -30255.782,E2 -30255.782} C_VEL
LIN {X 0,Y 61.26,Z 566.821,A -85,B 0,C 180,E1 -30258.836,E2 -30258.836} C_VEL
LIN {X 0,Y 53.557,Z 576.365,A -85,B 0,C 180,E1 -30263.285,E2 -30263.285} C_VEL
LIN {X 0,Y 47.573,Z 582.677,A -85,B 0,C 180,E1 -30267.581,E2 -30267.581} C_VEL
LIN {X 0,Y 39.555,Z 590.634,A -85,B 0,C 180,E1 -30276.916,E2 -30276.916} C_VEL
LIN {X 0,Y 32.828,Z 596.936,A -85,B 0,C 180,E1 -30290.04,E2 -30290.04} C_VEL
LIN {X 0,Y 28.573,Z 601.933,A -85,B 0,C 180,E1 -30308.35,E2 -30308.35} C_VEL
LIN {X 0,Y 27.551,Z 605.741,A -85,B 0,C 180,E1 -30330,E2 -30330} C_VEL
LIN {X 0,Y 27.954,Z 607.605,A -85,B 0,C 180,E1 -30344.561,E2 -30344.561} C_VEL
LIN {X 0,Y 29.762,Z 609.043,A -85,B 0,C 180,E1 -30358.182,E2 -30358.182} C_VEL
LIN {X 0,Y 32.975,Z 610.067,A -85,B 0,C 180,E1 -30369.745,E2 -30369.745} C_VEL
LIN {X 0,Y 42.387,Z 610.94,A -85,B 0,C 180,E1 -30385.997,E2 -30385.997} C_VEL
LIN {X 0,Y 53.977,Z 610.341,A -85,B 0,C 180,E1 -30395.7,E2 -30395.7} C_VEL
LIN {X 0,Y 66.57,Z 608.156,A -85,B 0,C 180,E1 -30401.83,E2 -30401.83} C_VEL
LIN {X 0,Y 79.711,Z 604.4,A -85,B 0,C 180,E1 -30405.889,E2 -30405.889} C_VEL
LIN {X 0,Y 89.791,Z 600.405,A -85,B 0,C 180,E1 -30408.058,E2 -30408.058} C_VEL
LIN {X 0,Y 100.004,Z 595.311,A -85,B 0,C 180,E1 -30409.692,E2 -30409.692} C_VEL
LIN {X 0,Y 110.291,Z 588.95,A -85,B 0,C 180,E1 -30410.993,E2 -30410.993} C_VEL
LIN {X 0,Y 120.636,Z 581.035,A -85,B 0,C 180,E1 -30412.04,E2 -30412.04} C_VEL
LIN {X 0,Y 127.561,Z 574.765,A -85,B 0,C 180,E1 -30412.608,E2 -30412.608} C_VEL
LIN {X 0,Y 127.38,Z 574.885,A -85,B 0,C 180,E1 -30413.265,E2 -30413.265} C_VEL
LIN {X 0,Y 118.305,Z 582.794,A -85,B 0,C 180,E1 -30414.28,E2 -30414.28} C_VEL
LIN {X 0,Y 107.472,Z 590.469,A -85,B 0,C 180,E1 -30415.739,E2 -30415.739} C_VEL
LIN {X 0,Y 98.511,Z 595.629,A -85,B 0,C 180,E1 -30417.156,E2 -30417.156} C_VEL
LIN {X 0,Y 87.502,Z 600.713,A -85,B 0,C 180,E1 -30419.373,E2 -30419.373} C_VEL
LIN {X 0,Y 77.351,Z 604.292,A -85,B 0,C 180,E1 -30421.954,E2 -30421.954} C_VEL
LIN {X 0,Y 65.184,Z 607.307,A -85,B 0,C 180,E1 -30426.225,E2 -30426.225} C_VEL
LIN {X 0,Y 57.115,Z 608.506,A -85,B 0,C 180,E1 -30430.142,E2 -30430.142} C_VEL
LIN {X 0,Y 46.953,Z 609.126,A -85,B 0,C 180,E1 -30437.422,E2 -30437.422} C_VEL
LIN {X 0,Y 39.709,Z 608.793,A -85,B 0,C 180,E1 -30445.48,E2 -30445.48} C_VEL
LIN {X 0,Y 35.199,Z 608.343,A -85,B 0,C 180,E1 -30451.282,E2 -30451.282} C_VEL
LIN {X 0,Y 27.362,Z 606.926,A -85,B 0,C 180,E1 -30462.205,E2 -30462.205} C_VEL
LIN {X 0,Y 22.078,Z 605.231,A -85,B 0,C 180,E1 -30475.6,E2 -30475.6} C_VEL
LIN {X 0,Y 19.985,Z 603.628,A -85,B 0,C 180,E1 -30490.164,E2 -30490.164} C_VEL
LIN {X 0,Y 19.864,Z 603.014,A -85,B 0,C 180,E1 -30495.589,E2 -30495.589} C_VEL
LIN {X 0,Y 23.348,Z 598.231,A -85,B 0,C 180,E1 -30527.518,E2 -30527.518} C_VEL
LIN {X 0,Y 30.089,Z 592.746,A -85,B 0,C 180,E1 -30545.727,E2 -30545.727} C_VEL
LIN {X 0,Y 38.431,Z 585.91,A -85,B 0,C 180,E1 -30557.01,E2 -30557.01} C_VEL
LIN {X 0,Y 46.231,Z 578.791,A -85,B 0,C 180,E1 -30563.311,E2 -30563.311} C_VEL
LIN {X 0,Y 53.996,Z 570.565,A -85,B 0,C 180,E1 -30567.781,E2 -30567.781} C_VEL
LIN {X 0,Y 62.106,Z 560.298,A -85,B 0,C 180,E1 -30571.28,E2 -30571.28} C_VEL
LIN {X 0,Y 68.792,Z 550.055,A -85,B 0,C 180,E1 -30573.368,E2 -30573.368} C_VEL
LIN {X 0,Y 74.621,Z 538.937,A -85,B 0,C 180,E1 -30575.025,E2 -30575.025} C_VEL
LIN {X 0,Y 79.351,Z 527.469,A -85,B 0,C 180,E1 -30576.135,E2 -30576.135} C_VEL
LIN {X 0,Y 83.149,Z 514.736,A -85,B 0,C 180,E1 -30577.062,E2 -30577.062} C_VEL
LIN {X 0,Y 85.758,Z 500.967,A -85,B 0,C 180,E1 -30577.62,E2 -30577.62} C_VEL
LIN {X 0,Y 87.178,Z 489.206,A -85,B 0,C 180,E1 -30578.011,E2 -30578.011} C_VEL
LIN {X 0,Y 86.202,Z 485.269,A -85,B 0,C 180,E1 -30583.114,E2 -30583.114} C_VEL
LIN {X 0,Y 85.888,Z 483.871,A -85,B 0,C 180,E1 -30585.788,E2 -30585.788} C_VEL
LIN {X 0,Y 85.629,Z 482.671,A -85,B 0,C 180,E1 -30590.551,E2 -30590.551} C_VEL
LIN {X 0,Y 85.796,Z 482.878,A -85,B 0,C 180,E1 -30595.874,E2 -30595.874} C_VEL
LIN {X 0,Y 86.02,Z 483.997,A -85,B 0,C 180,E1 -30598.499,E2 -30598.499} C_VEL
LIN {X 0,Y 86.774,Z 487.271,A -85,B 0,C 180,E1 -30603.372,E2 -30603.372} C_VEL
LIN {X 0,Y 87.255,Z 489.434,A -85,B 0,C 180,E1 -30605.61,E2 -30605.61} C_VEL
LIN {X 0,Y 84.572,Z 509.366,A -85,B 0,C 180,E1 -30606.223,E2 -30606.223} C_VEL
LIN {X 0,Y 81.36,Z 522.655,A -85,B 0,C 180,E1 -30606.818,E2 -30606.818} C_VEL
LIN {X 0,Y 77.117,Z 534.638,A -85,B 0,C 180,E1 -30607.664,E2 -30607.664} C_VEL
LIN {X 0,Y 72.008,Z 545.629,A -85,B 0,C 180,E1 -30608.818,E2 -30608.818} C_VEL
LIN {X 0,Y 66.033,Z 555.765,A -85,B 0,C 180,E1 -30610.109,E2 -30610.109} C_VEL
LIN {X 0,Y 58.507,Z 566.392,A -85,B 0,C 180,E1 -30612.584,E2 -30612.584} C_VEL
LIN {X 0,Y 51.163,Z 575.089,A -85,B 0,C 180,E1 -30615.944,E2 -30615.944} C_VEL
LIN {X 0,Y 44.694,Z 581.514,A -85,B 0,C 180,E1 -30619.36,E2 -30619.36} C_VEL
LIN {X 0,Y 35.716,Z 589.656,A -85,B 0,C 180,E1 -30627.693,E2 -30627.693} C_VEL
LIN {X 0,Y 27.732,Z 596.102,A -85,B 0,C 180,E1 -30640.512,E2 -30640.512} C_VEL
LIN {X 0,Y 22.085,Z 601.205,A -85,B 0,C 180,E1 -30661.49,E2 -30661.49} C_VEL
LIN {X 0,Y 20.449,Z 605.117,A -85,B 0,C 180,E1 -30690,E2 -30690} C_VEL
LIN {X 0,Y 21.149,Z 607.027,A -85,B 0,C 180,E1 -30709.409,E2 -30709.409} C_VEL
LIN {X 0,Y 27.866,Z 609.602,A -85,B 0,C 180,E1 -30739.165,E2 -30739.165} C_VEL
LIN {X 0,Y 33.018,Z 610.283,A -85,B 0,C 180,E1 -30748.363,E2 -30748.363} C_VEL
LIN {X 0,Y 45.028,Z 610.511,A -85,B 0,C 180,E1 -30759.465,E2 -30759.465} C_VEL
LIN {X 0,Y 58.028,Z 609.257,A -85,B 0,C 180,E1 -30765.671,E2 -30765.671} C_VEL
LIN {X 0,Y 71.461,Z 606.389,A -85,B 0,C 180,E1 -30769.563,E2 -30769.563} C_VEL
LIN {X 0,Y 81.713,Z 603.167,A -85,B 0,C 180,E1 -30771.524,E2 -30771.524} C_VEL
LIN {X 0,Y 92.049,Z 598.922,A -85,B 0,C 180,E1 -30772.994,E2 -30772.994} C_VEL
LIN {X 0,Y 91.89,Z 598.943,A -85,B 0,C 180,E1 -30773.854,E2 -30773.854} C_VEL
LIN {X 0,Y 80.624,Z 603.328,A -85,B 0,C 180,E1 -30775.775,E2 -30775.775} C_VEL
LIN {X 0,Y 70.317,Z 606.263,A -85,B 0,C 180,E1 -30778.093,E2 -30778.093} C_VEL
LIN {X 0,Y 63.251,Z 607.737,A -85,B 0,C 180,E1 -30780.118,E2 -30780.118} C_VEL
LIN {X 0,Y 56.281,Z 608.735,A -85,B 0,C 180,E1 -30782.615,E2 -30782.615} C_VEL
LIN {X 0,Y 44.001,Z 609.473,A -85,B 0,C 180,E1 -30789.193,E2 -30789.193} C_VEL
LIN {X 0,Y 35.145,Z 609.023,A -85,B 0,C 180,E1 -30797.158,E2 -30797.158} C_VEL
LIN {X 0,Y 25.58,Z 607.339,A -85,B 0,C 180,E1 -30814.491,E2 -30814.491} C_VEL
LIN {X 0,Y 20.53,Z 604.805,A -85,B 0,C 180,E1 -30839.105,E2 -30839.105} C_VEL
LIN {X 0,Y 19.864,Z 603.014,A -85,B 0,C 180,E1 -30855.589,E2 -30855.589} C_VEL
LIN {X 0,Y 20.033,Z 601.083,A -85,B 0,C 180,E1 -30871.65,E2 -30871.65} C_VEL
LIN {X 0,Y 20.652,Z 598.92,A -85,B 0,C 180,E1 -30887.237,E2 -30887.237} C_VEL
LIN {X 0,Y 25.972,Z 592.971,A -85,B 0,C 180,E1 -30915.935,E2 -30915.935} C_VEL
LIN {X 0,Y 30.019,Z 589.899,A -85,B 0,C 180,E1 -30922.351,E2 -30922.351} C_VEL
LIN {X 0,Y 40.524,Z 581.638,A -85,B 0,C 180,E1 -30930.125,E2 -30930.125} C_VEL
LIN {X 0,Y 49.662,Z 572.871,A -85,B 0,C 180,E1 -30934.39,E2 -30934.39} C_VEL
LIN {X 0,Y 57.312,Z 564.1,A -85,B 0,C 180,E1 -30936.88,E2 -30936.88} C_VEL
LIN {X 0,Y 65.025,Z 553.373,A -85,B 0,C 180,E1 -30938.777,E2 -30938.777} C_VEL
LIN {X 0,Y 71.054,Z 543.008,A -85,B 0,C 180,E1 -30939.99,E2 -30939.99} C_VEL
LIN {X 0,Y 76.36,Z 531.415,A -85,B 0,C 180,E1 -30940.972,E2 -30940.972} C_VEL
LIN {X 0,Y 80.625,Z 518.846,A -85,B 0,C 180,E1 -30941.667,E2 -30941.667} C_VEL
LIN {X 0,Y 83.635,Z 505.693,A -85,B 0,C 180,E1 -30942.191,E2 -30942.191} C_VEL
LIN {X 0,Y 85.29,Z 493.309,A -85,B 0,C 180,E1 -30942.617,E2 -30942.617} C_VEL
LIN {X 0,Y 84.905,Z 490.841,A -85,B 0,C 180,E1 -30946.536,E2 -30946.536} C_VEL
LIN {X 0,Y 84.732,Z 489.845,A -85,B 0,C 180,E1 -30950.45,E2 -30950.45} C_VEL
LIN {X 0,Y 84.855,Z 489.869,A -85,B 0,C 180,E1 -30955.248,E2 -30955.248} C_VEL
LIN {X 0,Y 85.126,Z 491.891,A -85,B 0,C 180,E1 -30959.089,E2 -30959.089} C_VEL
LIN {X 0,Y 85.375,Z 493.347,A -85,B 0,C 180,E1 -30961.111,E2 -30961.111} C_VEL
LIN {X 0,Y 83.044,Z 509.529,A -85,B 0,C 180,E1 -30961.476,E2 -30961.476} C_VEL
LIN {X 0,Y 79.846,Z 522.398,A -85,B 0,C 180,E1 -30961.888,E2 -30961.888} C_VEL
LIN {X 0,Y 75.619,Z 534.125,A -85,B 0,C 180,E1 -30962.465,E2 -30962.465} C_VEL
LIN {X 0,Y 70.392,Z 545.149,A -85,B 0,C 180,E1 -30963.254,E2 -30963.254} C_VEL
LIN {X 0,Y 64.291,Z 555.315,A -85,B 0,C 180,E1 -30964.066,E2 -30964.066} C_VEL
LIN {X 0,Y 58.245,Z 563.814,A -85,B 0,C 180,E1 -30965.476,E2 -30965.476} C_VEL
LIN {X 0,Y 49.674,Z 573.77,A -85,B 0,C 180,E1 -30967.968,E2 -30967.968} C_VEL
LIN {X 0,Y 41.185,Z 581.875,A -85,B 0,C 180,E1 -30971.132,E2 -30971.132} C_VEL
LIN {X 0,Y 31.403,Z 589.866,A -85,B 0,C 180,E1 -30977.988,E2 -30977.988} C_VEL
LIN {X 0,Y 23.712,Z 595.242,A -85,B 0,C 180,E1 -30987.232,E2 -30987.232} C_VEL
LIN {X 0,Y 16.182,Z 600.474,A -85,B 0,C 180,E1 -31009.348,E2 -31009.348} C_VEL
LIN {X 0,Y 13.367,Z 604.488,A -85,B 0,C 180,E1 -31050,E2 -31050} C_VEL
LIN {X 0,Y 14.638,Z 606.449,A -85,B 0,C 180,E1 -31078.693,E2 -31078.693} C_VEL
LIN {X 0,Y 23.826,Z 609.113,A -85,B 0,C 180,E1 -31112.24,E2 -31112.24} C_VEL
LIN {X 0,Y 29.902,Z 609.871,A -85,B 0,C 180,E1 -31120.069,E2 -31120.069} C_VEL
LIN {X 0,Y 43.048,Z 610.198,A -85,B 0,C 180,E1 -31128.386,E2 -31128.386} C_VEL
LIN {X 0,Y 56.685,Z 609.038,A -85,B 0,C 180,E1 -31132.673,E2 -31132.673} C_VEL
LIN {X 0,Y 58.937,Z 608.697,A -85,B 0,C 180,E1 -31133.153,E2 -31133.153} C_VEL
LIN {X 0,Y 56.435,Z 608.964,A -85,B 0,C 180,E1 -31135.025,E2 -31135.025} C_VEL
LIN {X 0,Y 49.256,Z 609.597,A -85,B 0,C 180,E1 -31137.14,E2 -31137.14} C_VEL
LIN {X 0,Y 42.071,Z 609.82,A -85,B 0,C 180,E1 -31140.002,E2 -31140.002} C_VEL
LIN {X 0,Y 35.221,Z 609.604,A -85,B 0,C 180,E1 -31143.905,E2 -31143.905} C_VEL
LIN {X 0,Y 28.505,Z 608.938,A -85,B 0,C 180,E1 -31149.529,E2 -31149.529} C_VEL
LIN {X 0,Y 22.225,Z 607.86,A -85,B 0,C 180,E1 -31158.44,E2 -31158.44} C_VEL
LIN {X 0,Y 16.79,Z 606.368,A -85,B 0,C 180,E1 -31173.16,E2 -31173.16} C_VEL
LIN {X 0,Y 12.776,Z 603.087,A -85,B 0,C 180,E1 -31216.029,E2 -31216.029} C_VEL
LIN {X 0,Y 16.569,Z 599.048,A -85,B 0,C 180,E1 -31255.097,E2 -31255.097} C_VEL
LIN {X 0,Y 26.095,Z 592.645,A -85,B 0,C 180,E1 -31277.785,E2 -31277.785} C_VEL
LIN {X 0,Y 30.019,Z 589.899,A -85,B 0,C 180,E1 -31282.351,E2 -31282.351} C_VEL
LIN {X 0,Y 34.144,Z 586.659,A -85,B 0,C 180,E1 -31287.195,E2 -31287.195} C_VEL
LIN {X 0,Y 40.316,Z 580.954,A -85,B 0,C 180,E1 -31295.432,E2 -31295.432} C_VEL
LIN {X 0,Y 46.617,Z 574.709,A -85,B 0,C 180,E1 -31301.354,E2 -31301.354} C_VEL
LIN {X 0,Y 50.609,Z 570.521,A -85,B 0,C 180,E1 -31302.902,E2 -31302.902} C_VEL
LIN {X 0,Y 59.274,Z 560.143,A -85,B 0,C 180,E1 -31304.438,E2 -31304.438} C_VEL
LIN {X 0,Y 66.307,Z 549.737,A -85,B 0,C 180,E1 -31305.275,E2 -31305.275} C_VEL
LIN {X 0,Y 72.432,Z 538.383,A -85,B 0,C 180,E1 -31305.993,E2 -31305.993} C_VEL
LIN {X 0,Y 77.613,Z 525.733,A -85,B 0,C 180,E1 -31306.469,E2 -31306.469} C_VEL
LIN {X 0,Y 81.562,Z 511.93,A -85,B 0,C 180,E1 -31306.889,E2 -31306.889} C_VEL
LIN {X 0,Y 83.846,Z 498.647,A -85,B 0,C 180,E1 -31307.163,E2 -31307.163} C_VEL
LIN {X 0,Y 83.919,Z 497.913,A -85,B 0,C 180,E1 -31307.346,E2 -31307.346} C_VEL
LIN {X 0,Y 83.838,Z 496.988,A -85,B 0,C 180,E1 -31310.347,E2 -31310.347} C_VEL
LIN {X 0,Y 83.939,Z 497.354,A -85,B 0,C 180,E1 -31315.562,E2 -31315.562} C_VEL
LIN {X 0,Y 83.959,Z 497.864,A -85,B 0,C 180,E1 -31316.364,E2 -31316.364} C_VEL
LIN {X 0,Y 81.792,Z 511.292,A -85,B 0,C 180,E1 -31316.611,E2 -31316.611} C_VEL
LIN {X 0,Y 78.191,Z 524.423,A -85,B 0,C 180,E1 -31316.882,E2 -31316.882} C_VEL
LIN {X 0,Y 73.886,Z 535.595,A -85,B 0,C 180,E1 -31317.116,E2 -31317.116} C_VEL
LIN {X 0,Y 67.703,Z 547.853,A -85,B 0,C 180,E1 -31317.587,E2 -31317.587} C_VEL
LIN {X 0,Y 60.656,Z 558.672,A -85,B 0,C 180,E1 -31317.904,E2 -31317.904} C_VEL
LIN {X 0,Y 52.716,Z 568.615,A -85,B 0,C 180,E1 -31319.033,E2 -31319.033} C_VEL
LIN {X 0,Y 44.974,Z 576.629,A -85,B 0,C 180,E1 -31320.333,E2 -31320.333} C_VEL
LIN {X 0,Y 36.921,Z 583.639,A -85,B 0,C 180,E1 -31322.109,E2 -31322.109} C_VEL
LIN {X 0,Y 26.525,Z 591.177,A -85,B 0,C 180,E1 -31326.502,E2 -31326.502} C_VEL
LIN {X 0,Y 14.812,Z 598.069,A -85,B 0,C 180,E1 -31338.39,E2 -31338.39} C_VEL
LIN {X 0,Y 6.919,Z 602.582,A -85,B 0,C 180,E1 -31379.478,E2 -31379.478} C_VEL
LIN {X 0,Y 6.27,Z 603.824,A -85,B 0,C 180,E1 -31410,E2 -31410} C_VEL
LIN {X 0,Y 9.078,Z 605.872,A -85,B 0,C 180,E1 -31460.729,E2 -31460.729} C_VEL
LIN {X 0,Y 21.456,Z 608.625,A -85,B 0,C 180,E1 -31489.308,E2 -31489.308} C_VEL
LIN {X 0,Y 28.279,Z 609.429,A -85,B 0,C 180,E1 -31493.767,E2 -31493.767} C_VEL
LIN {X 0,Y 28.246,Z 609.41,A -85,B 0,C 180,E1 -31494.409,E2 -31494.409} C_VEL
LIN {X 0,Y 19.81,Z 608.157,A -85,B 0,C 180,E1 -31500.005,E2 -31500.005} C_VEL
LIN {X 0,Y 8.027,Z 605.048,A -85,B 0,C 180,E1 -31528.888,E2 -31528.888} C_VEL
LIN {X 0,Y 8.3,Z 600.939,A -85,B 0,C 180,E1 -31622.118,E2 -31622.118} C_VEL
LIN {X 0,Y 16.844,Z 596.461,A -85,B 0,C 180,E1 -31646.558,E2 -31646.558} C_VEL
LIN {X 0,Y 27.546,Z 590.033,A -85,B 0,C 180,E1 -31655.644,E2 -31655.644} C_VEL
LIN {X 0,Y 37.467,Z 582.772,A -85,B 0,C 180,E1 -31659.696,E2 -31659.696} C_VEL
LIN {X 0,Y 46.771,Z 574.483,A -85,B 0,C 180,E1 -31662.203,E2 -31662.203} C_VEL
LIN {X 0,Y 50.609,Z 570.521,A -85,B 0,C 180,E1 -31662.902,E2 -31662.902} C_VEL
LIN {X 0,Y 50.129,Z 570.927,A -85,B 0,C 180,E1 -31664.104,E2 -31664.104} C_VEL
LIN {X 0,Y 46.108,Z 574.832,A -85,B 0,C 180,E1 -31666.946,E2 -31666.946} C_VEL
LIN {X 0,Y 39.809,Z 580.505,A -85,B 0,C 180,E1 -31670.011,E2 -31670.011} C_VEL
LIN {X 0,Y 35.342,Z 584.111,A -85,B 0,C 180,E1 -31671.022,E2 -31671.022} C_VEL
LIN {X 0,Y 28.447,Z 589.098,A -85,B 0,C 180,E1 -31671.186,E2 -31671.186} C_VEL
LIN {X 0,Y 28.497,Z 589.055,A -85,B 0,C 180,E1 -31670.566,E2 -31670.566} C_VEL
LIN {X 0,Y 39.176,Z 581.03,A -85,B 0,C 180,E1 -31670.625,E2 -31670.625} C_VEL
LIN {X 0,Y 48.717,Z 572.18,A -85,B 0,C 180,E1 -31670.954,E2 -31670.954} C_VEL
LIN {X 0,Y 56.871,Z 562.943,A -85,B 0,C 180,E1 -31671.343,E2 -31671.343} C_VEL
LIN {X 0,Y 48.661,Z 572.247,A -85,B 0,C 180,E1 -31671.376,E2 -31671.376} C_VEL
LIN {X 0,Y 39.14,Z 581.067,A -85,B 0,C 180,E1 -31670.95,E2 -31670.95} C_VEL
LIN {X 0,Y 35.342,Z 584.111,A -85,B 0,C 180,E1 -31671.022,E2 -31671.022} C_VEL
LIN {X 0,Y 34.568,Z 585.692,A -85,B 0,C 180,E1 -31671.033,E2 -31671.033} C_VEL
LIN {X 0,Y 34.568,Z 600,A -85,B 0,C 180,E1 -31671.033,E2 -31671.033} C_VEL
LIN {X 0,Y 34.568,Z 600,A -85,B 0,C 180,E1 -31671.033,E2 -31671.033}

QRS_NEXT_CUT()

QRS_NEXT()
QRS_HOME()

END
